KUKA KRL program: EPS_2_25862_MH02_A_20251016040656.src

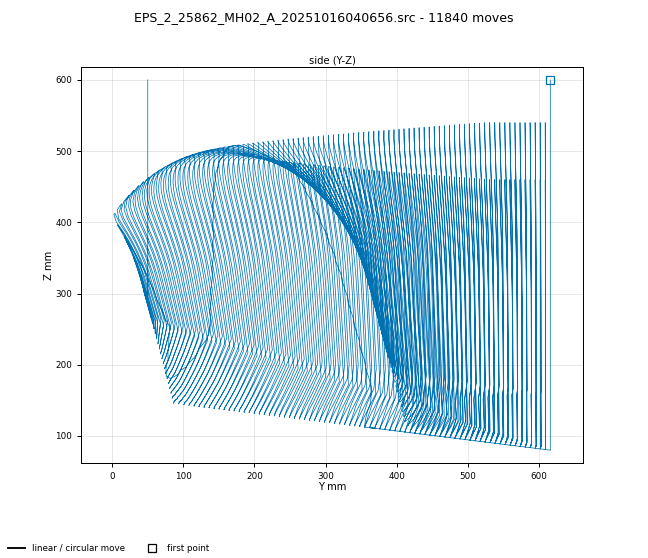
[picture p0: tool path of EPS_2_25862_MH02_A_20251016040656.src, 11840 of 11842 moves have a stored position in this frame; points joined in program order, loops and branches not executed]
&ACCESS RVP
&REL 4
&COMMENT QRS 19112012
&PARAM EDITMASK = *
DEF PART()
EXT BAS (BAS_COMMAND :IN,REAL :IN )
INT I
BAS (#INITMOV,0 )

;KUKA QRS Post kuka4.cps  Date:22-06-2017 !

File_ID=2894

QRS_PRE_INIT()

;Init var - Until changes are made in qrs_pre_init
Outlet_Square_prg=0
Inlet_1_Square_prg=0
Inlet_2_Square_prg=0
Inlet_3_Square_prg=0
Inlet_4_Square_prg=0
Inlet_5_Square_prg=0

Outlet_1={X 0.000, Y 524.050, Z 357.000, B 0.000, E1 0.000 }
Inlet_1={X 0.000, Y 530.010, Z 277.000, B 0.000, E1 270.000 }
Outlet_1_type=366
Inlet_1_type=366
;QRS#1=Sidecore dimensions
;QRS#2=375-15" PVC SDR 35
;QRS#3=375-15" PVC SDR 35
;QRS#4=
;QRS#5=
;QRS#6=
;QRS#7=
;QRS#8=
;QRS#9=20Y PSX
;QRS#10=20Y PSX
;QRS#11=
;QRS#12=
;QRS#13=
;QRS#14=
;QRS#15=
;QRS#16=1220x127x838 2,75'
;QRS#17=EPS Height
;QRS#18=540
;QRS#19=*
;QRS#20= UPDATED VERSION 22-06-2017
;QRS#21=*
Outlet_Square=0250
Inlet_1_Square=0250
Inlet_2_Square=0
Inlet_3_Square=0
Inlet_4_Square=0
Inlet_5_Square=0
Mill_Square=1
Outlet_Square_Prg=252
Inlet_1_Square_prg=252

QRS_INIT()

$ADVANCE=5

; T1
PTP {E1 173.606,E2 173.606}
PTP {X 0,Y 615.5,A -85,B 0,C 180,E1 173.606,E2 173.606,E3 0,E4 0,E5 0,E6 0}
QRS_SPEED_INIT()
LIN {X 0,Y 615.5,Z 600,A -85,B 0,C 180,E1 173.606,E2 173.606,E3 0,E4 0,E5 0,E6 0} C_VEL
LIN {X 0,Y 615.5,Z 90.176,A -85,B 0,C 180,E1 173.606,E2 173.606} C_VEL
LIN {X 0,Y 615.5,Z 81.996,A -85,B 0,C 180,E1 173.606,E2 173.606} C_VEL
LIN {X 0,Y 615.484,Z 79.996,A -85,B 0,C 180,E1 173.42,E2 173.42} C_VEL
LIN {X 0,Y 615.476,Z 80.009,A -85,B 0,C 180,E1 170.801,E2 170.801} C_VEL
LIN {X 0,Y 615.482,Z 80.003,A -85,B 0,C 180,E1 168.139,E2 168.139} C_VEL
LIN {X 0,Y 615.478,Z 79.998,A -85,B 0,C 180,E1 165.451,E2 165.451} C_VEL
LIN {X 0,Y 615.495,Z 80.012,A -85,B 0,C 180,E1 162.73,E2 162.73} C_VEL
LIN {X 0,Y 615.491,Z 79.995,A -85,B 0,C 180,E1 159.967,E2 159.967} C_VEL
LIN {X 0,Y 615.473,Z 80.006,A -85,B 0,C 180,E1 157.155,E2 157.155} C_VEL
LIN {X 0,Y 615.483,Z 80.004,A -85,B 0,C 180,E1 154.431,E2 154.431} C_VEL
LIN {X 0,Y 615.484,Z 79.997,A -85,B 0,C 180,E1 152.085,E2 152.085} C_VEL
LIN {X 0,Y 615.486,Z 79.995,A -85,B 0,C 180,E1 149.84,E2 149.84} C_VEL
LIN {X 0,Y 615.473,Z 80.002,A -85,B 0,C 180,E1 147.542,E2 147.542} C_VEL
LIN {X 0,Y 615.483,Z 80.009,A -85,B 0,C 180,E1 145.185,E2 145.185} C_VEL
LIN {X 0,Y 615.485,Z 80.007,A -85,B 0,C 180,E1 142.758,E2 142.758} C_VEL
LIN {X 0,Y 615.481,Z 79.997,A -85,B 0,C 180,E1 139.911,E2 139.911} C_VEL
LIN {X 0,Y 615.473,Z 80.003,A -85,B 0,C 180,E1 137.646,E2 137.646} C_VEL
LIN {X 0,Y 615.486,Z 80.008,A -85,B 0,C 180,E1 134.931,E2 134.931} C_VEL
LIN {X 0,Y 615.483,Z 79.996,A -85,B 0,C 180,E1 132.08,E2 132.08} C_VEL
LIN {X 0,Y 615.473,Z 80.003,A -85,B 0,C 180,E1 129.751,E2 129.751} C_VEL
LIN {X 0,Y 615.482,Z 80.005,A -85,B 0,C 180,E1 126.936,E2 126.936} C_VEL
LIN {X 0,Y 615.473,Z 80,A -85,B 0,C 180,E1 124.022,E2 124.022} C_VEL
LIN {X 0,Y 615.479,Z 80.007,A -85,B 0,C 180,E1 121.685,E2 121.685} C_VEL
LIN {X 0,Y 615.491,Z 80.014,A -85,B 0,C 180,E1 119.406,E2 119.406} C_VEL
LIN {X 0,Y 615.485,Z 79.995,A -85,B 0,C 180,E1 116.444,E2 116.444} C_VEL
LIN {X 0,Y 615.485,Z 80.015,A -85,B 0,C 180,E1 113.556,E2 113.556} C_VEL
LIN {X 0,Y 615.485,Z 79.996,A -85,B 0,C 180,E1 110.556,E2 110.556} C_VEL
LIN {X 0,Y 615.475,Z 80.007,A -85,B 0,C 180,E1 107.957,E2 107.957} C_VEL
LIN {X 0,Y 615.481,Z 80.003,A -85,B 0,C 180,E1 105.226,E2 105.226} C_VEL
LIN {X 0,Y 615.481,Z 79.997,A -85,B 0,C 180,E1 102.53,E2 102.53} C_VEL
LIN {X 0,Y 615.492,Z 80.011,A -85,B 0,C 180,E1 99.862,E2 99.862} C_VEL
LIN {X 0,Y 615.482,Z 80,A -85,B 0,C 180,E1 97.215,E2 97.215} C_VEL
LIN {X 0,Y 615.478,Z 79.999,A -85,B 0,C 180,E1 94.584,E2 94.584} C_VEL
LIN {X 0,Y 615.495,Z 80.012,A -85,B 0,C 180,E1 91.963,E2 91.963} C_VEL
LIN {X 0,Y 615.482,Z 79.999,A -85,B 0,C 180,E1 89.345,E2 89.345} C_VEL
LIN {X 0,Y 615.479,Z 79.999,A -85,B 0,C 180,E1 86.727,E2 86.727} C_VEL
LIN {X 0,Y 615.493,Z 80.012,A -85,B 0,C 180,E1 84.101,E2 84.101} C_VEL
LIN {X 0,Y 615.482,Z 79.999,A -85,B 0,C 180,E1 81.463,E2 81.463} C_VEL
LIN {X 0,Y 615.477,Z 80,A -85,B 0,C 180,E1 78.806,E2 78.806} C_VEL
LIN {X 0,Y 615.491,Z 80.01,A -85,B 0,C 180,E1 76.066,E2 76.066} C_VEL
LIN {X 0,Y 615.49,Z 79.995,A -85,B 0,C 180,E1 73.413,E2 73.413} C_VEL
LIN {X 0,Y 615.477,Z 80.005,A -85,B 0,C 180,E1 70.661,E2 70.661} C_VEL
LIN {X 0,Y 615.479,Z 80.003,A -85,B 0,C 180,E1 67.863,E2 67.863} C_VEL
LIN {X 0,Y 615.477,Z 80,A -85,B 0,C 180,E1 65.007,E2 65.007} C_VEL
LIN {X 0,Y 615.477,Z 80.005,A -85,B 0,C 180,E1 62.822,E2 62.822} C_VEL
LIN {X 0,Y 615.483,Z 80.007,A -85,B 0,C 180,E1 60.206,E2 60.206} C_VEL
LIN {X 0,Y 615.493,Z 79.994,A -85,B 0,C 180,E1 57.542,E2 57.542} C_VEL
LIN {X 0,Y 615.477,Z 80,A -85,B 0,C 180,E1 55.184,E2 55.184} C_VEL
LIN {X 0,Y 615.486,Z 80.01,A -85,B 0,C 180,E1 52.757,E2 52.757} C_VEL
LIN {X 0,Y 615.482,Z 79.998,A -85,B 0,C 180,E1 49.912,E2 49.912} C_VEL
LIN {X 0,Y 615.495,Z 79.993,A -85,B 0,C 180,E1 47.647,E2 47.647} C_VEL
LIN {X 0,Y 615.48,Z 80.01,A -85,B 0,C 180,E1 44.93,E2 44.93} C_VEL
LIN {X 0,Y 615.481,Z 79.998,A -85,B 0,C 180,E1 42.079,E2 42.079} C_VEL
LIN {X 0,Y 615.49,Z 79.995,A -85,B 0,C 180,E1 39.75,E2 39.75} C_VEL
LIN {X 0,Y 615.484,Z 80.014,A -85,B 0,C 180,E1 36.936,E2 36.936} C_VEL
LIN {X 0,Y 615.487,Z 79.995,A -85,B 0,C 180,E1 34.022,E2 34.022} C_VEL
LIN {X 0,Y 615.482,Z 80.012,A -85,B 0,C 180,E1 31.084,E2 31.084} C_VEL
LIN {X 0,Y 615.478,Z 80.001,A -85,B 0,C 180,E1 28.448,E2 28.448} C_VEL
LIN {X 0,Y 615.478,Z 80,A -85,B 0,C 180,E1 25.716,E2 25.716} C_VEL
LIN {X 0,Y 615.474,Z 80.004,A -85,B 0,C 180,E1 23.557,E2 23.557} C_VEL
LIN {X 0,Y 615.491,Z 80.049,A -85,B 0,C 180,E1 22.026,E2 22.026} C_VEL
LIN {X 0,Y 615.487,Z 80.696,A -85,B 0,C 180,E1 21.96,E2 21.96} C_VEL
LIN {X 0,Y 615.489,Z 286.31,A -85,B 0,C 180,E1 19.425,E2 19.425} C_VEL
LIN {X 0,Y 615.49,Z 302.93,A -85,B 0,C 180,E1 19.078,E2 19.078} C_VEL
LIN {X 0,Y 615.495,Z 319.071,A -85,B 0,C 180,E1 18.606,E2 18.606} C_VEL
LIN {X 0,Y 615.496,Z 334.183,A -85,B 0,C 180,E1 18.038,E2 18.038} C_VEL
LIN {X 0,Y 615.496,Z 348.835,A -85,B 0,C 180,E1 17.356,E2 17.356} C_VEL
LIN {X 0,Y 615.497,Z 363.769,A -85,B 0,C 180,E1 16.51,E2 16.51} C_VEL
LIN {X 0,Y 615.496,Z 377.743,A -85,B 0,C 180,E1 15.565,E2 15.565} C_VEL
LIN {X 0,Y 615.497,Z 390.512,A -85,B 0,C 180,E1 14.549,E2 14.549} C_VEL
LIN {X 0,Y 615.499,Z 401.486,A -85,B 0,C 180,E1 13.537,E2 13.537} C_VEL
LIN {X 0,Y 615.497,Z 412.376,A -85,B 0,C 180,E1 12.362,E2 12.362} C_VEL
LIN {X 0,Y 615.492,Z 422.792,A -85,B 0,C 180,E1 11.041,E2 11.041} C_VEL
LIN {X 0,Y 615.492,Z 431.704,A -85,B 0,C 180,E1 9.696,E2 9.696} C_VEL
LIN {X 0,Y 615.489,Z 438.268,A -85,B 0,C 180,E1 8.537,E2 8.537} C_VEL
LIN {X 0,Y 615.495,Z 445.804,A -85,B 0,C 180,E1 6.896,E2 6.896} C_VEL
LIN {X 0,Y 615.495,Z 451.596,A -85,B 0,C 180,E1 5.241,E2 5.241} C_VEL
LIN {X 0,Y 615.492,Z 454.979,A -85,B 0,C 180,E1 3.929,E2 3.929} C_VEL
LIN {X 0,Y 615.49,Z 457.428,A -85,B 0,C 180,E1 2.618,E2 2.618} C_VEL
LIN {X 0,Y 615.491,Z 458.838,A -85,B 0,C 180,E1 1.309,E2 1.309} C_VEL
LIN {X 0,Y 615.49,Z 459.385,A -85,B 0,C 180,E1 0,E2 0} C_VEL
LIN {X 0,Y 615.489,Z 458.902,A -85,B 0,C 180,E1 -1.309,E2 -1.309} C_VEL
LIN {X 0,Y 615.492,Z 457.568,A -85,B 0,C 180,E1 -2.618,E2 -2.618} C_VEL
LIN {X 0,Y 615.491,Z 455.174,A -85,B 0,C 180,E1 -3.928,E2 -3.928} C_VEL
LIN {X 0,Y 615.49,Z 451.879,A -85,B 0,C 180,E1 -5.241,E2 -5.241} C_VEL
LIN {X 0,Y 615.492,Z 446.153,A -85,B 0,C 180,E1 -6.898,E2 -6.898} C_VEL
LIN {X 0,Y 615.493,Z 440.328,A -85,B 0,C 180,E1 -8.206,E2 -8.206} C_VEL
LIN {X 0,Y 615.489,Z 432.251,A -85,B 0,C 180,E1 -9.696,E2 -9.696} C_VEL
LIN {X 0,Y 615.493,Z 423.461,A -85,B 0,C 180,E1 -11.041,E2 -11.041} C_VEL
LIN {X 0,Y 615.498,Z 413.171,A -85,B 0,C 180,E1 -12.362,E2 -12.362} C_VEL
LIN {X 0,Y 615.495,Z 402.356,A -85,B 0,C 180,E1 -13.537,E2 -13.537} C_VEL
LIN {X 0,Y 615.496,Z 391.545,A -85,B 0,C 180,E1 -14.549,E2 -14.549} C_VEL
LIN {X 0,Y 615.497,Z 377.814,A -85,B 0,C 180,E1 -15.65,E2 -15.65} C_VEL
LIN {X 0,Y 615.498,Z 363.993,A -85,B 0,C 180,E1 -16.586,E2 -16.586} C_VEL
LIN {X 0,Y 615.492,Z 348.926,A -85,B 0,C 180,E1 -17.442,E2 -17.442} C_VEL
LIN {X 0,Y 615.487,Z 332.529,A -85,B 0,C 180,E1 -18.2,E2 -18.2} C_VEL
LIN {X 0,Y 615.489,Z 316.698,A -85,B 0,C 180,E1 -18.775,E2 -18.775} C_VEL
LIN {X 0,Y 615.499,Z 301.255,A -85,B 0,C 180,E1 -19.207,E2 -19.207} C_VEL
LIN {X 0,Y 615.49,Z 285.06,A -85,B 0,C 180,E1 -19.533,E2 -19.533} C_VEL
LIN {X 0,Y 615.419,Z 80.715,A -85,B 0,C 180,E1 -22.051,E2 -22.051} C_VEL
LIN {X 0,Y 615.418,Z 80.012,A -85,B 0,C 180,E1 -22.139,E2 -22.139} C_VEL
LIN {X 0,Y 615.489,Z 80.013,A -85,B 0,C 180,E1 -24.992,E2 -24.992} C_VEL
LIN {X 0,Y 615.48,Z 80.009,A -85,B 0,C 180,E1 -27.177,E2 -27.177} C_VEL
LIN {X 0,Y 615.429,Z 80.01,A -85,B 0,C 180,E1 -29.784,E2 -29.784} C_VEL
LIN {X 0,Y 615.434,Z 80.008,A -85,B 0,C 180,E1 -31.688,E2 -31.688} C_VEL
LIN {X 0,Y 615.442,Z 80.009,A -85,B 0,C 180,E1 -34.025,E2 -34.025} C_VEL
LIN {X 0,Y 615.478,Z 80.014,A -85,B 0,C 180,E1 -36.425,E2 -36.425} C_VEL
LIN {X 0,Y 615.476,Z 80.001,A -85,B 0,C 180,E1 -39.06,E2 -39.06} C_VEL
LIN {X 0,Y 615.453,Z 80.005,A -85,B 0,C 180,E1 -41.476,E2 -41.476} C_VEL
LIN {X 0,Y 615.494,Z 80.014,A -85,B 0,C 180,E1 -44.149,E2 -44.149} C_VEL
LIN {X 0,Y 615.478,Z 79.998,A -85,B 0,C 180,E1 -46.953,E2 -46.953} C_VEL
LIN {X 0,Y 615.467,Z 80.005,A -85,B 0,C 180,E1 -49.392,E2 -49.392} C_VEL
LIN {X 0,Y 615.489,Z 80.008,A -85,B 0,C 180,E1 -51.988,E2 -51.988} C_VEL
LIN {X 0,Y 615.487,Z 79.998,A -85,B 0,C 180,E1 -54.384,E2 -54.384} C_VEL
LIN {X 0,Y 615.485,Z 79.997,A -85,B 0,C 180,E1 -56.763,E2 -56.763} C_VEL
LIN {X 0,Y 615.481,Z 80.005,A -85,B 0,C 180,E1 -59.08,E2 -59.08} C_VEL
LIN {X 0,Y 615.482,Z 80.01,A -85,B 0,C 180,E1 -61.55,E2 -61.55} C_VEL
LIN {X 0,Y 615.477,Z 80.197,A -85,B 0,C 180,E1 -62.153,E2 -62.153} C_VEL
LIN {X 0,Y 615.495,Z 116.189,A -85,B 0,C 180,E1 -64.864,E2 -64.864} C_VEL
LIN {X 0,Y 615.439,Z 150.773,A -85,B 0,C 180,E1 -67.409,E2 -67.409} C_VEL
LIN {X 0,Y 615.455,Z 158.788,A -85,B 0,C 180,E1 -67.972,E2 -67.972} C_VEL
LIN {X 0,Y 615.495,Z 366.404,A -85,B 0,C 180,E1 -70.532,E2 -70.532} C_VEL
LIN {X 0,Y 615.493,Z 382.979,A -85,B 0,C 180,E1 -70.878,E2 -70.878} C_VEL
LIN {X 0,Y 615.493,Z 397.921,A -85,B 0,C 180,E1 -71.311,E2 -71.311} C_VEL
LIN {X 0,Y 615.491,Z 413.342,A -85,B 0,C 180,E1 -71.88,E2 -71.88} C_VEL
LIN {X 0,Y 615.493,Z 427.997,A -85,B 0,C 180,E1 -72.558,E2 -72.558} C_VEL
LIN {X 0,Y 615.5,Z 441.829,A -85,B 0,C 180,E1 -73.328,E2 -73.328} C_VEL
LIN {X 0,Y 615.499,Z 456.032,A -85,B 0,C 180,E1 -74.265,E2 -74.265} C_VEL
LIN {X 0,Y 615.498,Z 469.087,A -85,B 0,C 180,E1 -75.282,E2 -75.282} C_VEL
LIN {X 0,Y 615.492,Z 480.209,A -85,B 0,C 180,E1 -76.294,E2 -76.294} C_VEL
LIN {X 0,Y 615.494,Z 491.287,A -85,B 0,C 180,E1 -77.47,E2 -77.47} C_VEL
LIN {X 0,Y 615.494,Z 500.763,A -85,B 0,C 180,E1 -78.64,E2 -78.64} C_VEL
LIN {X 0,Y 615.494,Z 509.962,A -85,B 0,C 180,E1 -79.971,E2 -79.971} C_VEL
LIN {X 0,Y 615.49,Z 518.499,A -85,B 0,C 180,E1 -81.463,E2 -81.463} C_VEL
LIN {X 0,Y 615.492,Z 525.981,A -85,B 0,C 180,E1 -83.102,E2 -83.102} C_VEL
LIN {X 0,Y 615.496,Z 531.739,A -85,B 0,C 180,E1 -84.758,E2 -84.758} C_VEL
LIN {X 0,Y 615.49,Z 535.076,A -85,B 0,C 180,E1 -86.071,E2 -86.071} C_VEL
LIN {X 0,Y 615.488,Z 537.503,A -85,B 0,C 180,E1 -87.382,E2 -87.382} C_VEL
LIN {X 0,Y 615.493,Z 538.869,A -85,B 0,C 180,E1 -88.691,E2 -88.691} C_VEL
LIN {X 0,Y 615.489,Z 539.39,A -85,B 0,C 180,E1 -90,E2 -90} C_VEL
LIN {X 0,Y 615.493,Z 538.869,A -85,B 0,C 180,E1 -91.308,E2 -91.308} C_VEL
LIN {X 0,Y 615.488,Z 537.504,A -85,B 0,C 180,E1 -92.617,E2 -92.617} C_VEL
LIN {X 0,Y 615.49,Z 535.078,A -85,B 0,C 180,E1 -93.928,E2 -93.928} C_VEL
LIN {X 0,Y 615.496,Z 531.742,A -85,B 0,C 180,E1 -95.241,E2 -95.241} C_VEL
LIN {X 0,Y 615.491,Z 525.983,A -85,B 0,C 180,E1 -96.898,E2 -96.898} C_VEL
LIN {X 0,Y 615.49,Z 518.504,A -85,B 0,C 180,E1 -98.536,E2 -98.536} C_VEL
LIN {X 0,Y 615.494,Z 509.967,A -85,B 0,C 180,E1 -100.028,E2 -100.028} C_VEL
LIN {X 0,Y 615.494,Z 500.77,A -85,B 0,C 180,E1 -101.359,E2 -101.359} C_VEL
LIN {X 0,Y 615.495,Z 491.295,A -85,B 0,C 180,E1 -102.529,E2 -102.529} C_VEL
LIN {X 0,Y 615.493,Z 480.219,A -85,B 0,C 180,E1 -103.705,E2 -103.705} C_VEL
LIN {X 0,Y 615.499,Z 468.12,A -85,B 0,C 180,E1 -104.802,E2 -104.802} C_VEL
LIN {X 0,Y 615.497,Z 454.884,A -85,B 0,C 180,E1 -105.819,E2 -105.819} C_VEL
LIN {X 0,Y 615.5,Z 441.844,A -85,B 0,C 180,E1 -106.671,E2 -106.671} C_VEL
LIN {X 0,Y 615.493,Z 428.015,A -85,B 0,C 180,E1 -107.441,E2 -107.441} C_VEL
LIN {X 0,Y 615.491,Z 413.357,A -85,B 0,C 180,E1 -108.119,E2 -108.119} C_VEL
LIN {X 0,Y 615.493,Z 397.948,A -85,B 0,C 180,E1 -108.688,E2 -108.688} C_VEL
LIN {X 0,Y 615.498,Z 381.192,A -85,B 0,C 180,E1 -109.164,E2 -109.164} C_VEL
LIN {X 0,Y 615.495,Z 364.975,A -85,B 0,C 180,E1 -109.489,E2 -109.489} C_VEL
LIN {X 0,Y 615.453,Z 158.208,A -85,B 0,C 180,E1 -112.049,E2 -112.049} C_VEL
LIN {X 0,Y 615.46,Z 124.216,A -85,B 0,C 180,E1 -114.542,E2 -114.542} C_VEL
LIN {X 0,Y 615.484,Z 89.011,A -85,B 0,C 180,E1 -117.177,E2 -117.177} C_VEL
LIN {X 0,Y 615.475,Z 79.998,A -85,B 0,C 180,E1 -117.869,E2 -117.869} C_VEL
LIN {X 0,Y 615.469,Z 80.004,A -85,B 0,C 180,E1 -120.161,E2 -120.161} C_VEL
LIN {X 0,Y 615.484,Z 80.01,A -85,B 0,C 180,E1 -122.457,E2 -122.457} C_VEL
LIN {X 0,Y 615.487,Z 80.008,A -85,B 0,C 180,E1 -124.814,E2 -124.814} C_VEL
LIN {X 0,Y 615.487,Z 79.997,A -85,B 0,C 180,E1 -127.242,E2 -127.242} C_VEL
LIN {X 0,Y 615.469,Z 80.006,A -85,B 0,C 180,E1 -130.087,E2 -130.087} C_VEL
LIN {X 0,Y 615.489,Z 80.011,A -85,B 0,C 180,E1 -132.352,E2 -132.352} C_VEL
LIN {X 0,Y 615.483,Z 79.998,A -85,B 0,C 180,E1 -135.068,E2 -135.068} C_VEL
LIN {X 0,Y 615.471,Z 80.005,A -85,B 0,C 180,E1 -137.921,E2 -137.921} C_VEL
LIN {X 0,Y 615.493,Z 80.011,A -85,B 0,C 180,E1 -140.251,E2 -140.251} C_VEL
LIN {X 0,Y 615.485,Z 79.996,A -85,B 0,C 180,E1 -143.063,E2 -143.063} C_VEL
LIN {X 0,Y 615.482,Z 79.996,A -85,B 0,C 180,E1 -145.299,E2 -145.299} C_VEL
LIN {X 0,Y 615.467,Z 80.004,A -85,B 0,C 180,E1 -147.671,E2 -147.671} C_VEL
LIN {X 0,Y 615.496,Z 80.011,A -85,B 0,C 180,E1 -150.203,E2 -150.203} C_VEL
LIN {X 0,Y 615.497,Z 79.993,A -85,B 0,C 180,E1 -152.952,E2 -152.952} C_VEL
LIN {X 0,Y 615.476,Z 80.007,A -85,B 0,C 180,E1 -155.728,E2 -155.728} C_VEL
LIN {X 0,Y 615.483,Z 80,A -85,B 0,C 180,E1 -158.568,E2 -158.568} C_VEL
LIN {X 0,Y 615.47,Z 80.003,A -85,B 0,C 180,E1 -161.398,E2 -161.398} C_VEL
LIN {X 0,Y 615.489,Z 80.008,A -85,B 0,C 180,E1 -164.095,E2 -164.095} C_VEL
LIN {X 0,Y 615.493,Z 79.994,A -85,B 0,C 180,E1 -166.799,E2 -166.799} C_VEL
LIN {X 0,Y 615.473,Z 80.007,A -85,B 0,C 180,E1 -169.473,E2 -169.473} C_VEL
LIN {X 0,Y 615.484,Z 80.004,A -85,B 0,C 180,E1 -172.124,E2 -172.124} C_VEL
LIN {X 0,Y 615.485,Z 79.995,A -85,B 0,C 180,E1 -174.759,E2 -174.759} C_VEL
LIN {X 0,Y 615.478,Z 80.007,A -85,B 0,C 180,E1 -177.382,E2 -177.382} C_VEL
LIN {X 0,Y 615.483,Z 80.004,A -85,B 0,C 180,E1 -180,E2 -180} C_VEL
LIN {X 0,Y 615.486,Z 79.995,A -85,B 0,C 180,E1 -182.618,E2 -182.618} C_VEL
LIN {X 0,Y 615.474,Z 80.008,A -85,B 0,C 180,E1 -185.241,E2 -185.241} C_VEL
LIN {X 0,Y 615.484,Z 79.996,A -85,B 0,C 180,E1 -186.58,E2 -186.58} C_VEL
LIN {X 0,Y 614.804,Z 80.154,A -85,B 0,C 180,E1 -187.126,E2 -187.126} C_VEL
LIN {X 0,Y 611.965,Z 80.565,A -85,B 0,C 180,E1 -188.012,E2 -188.012} C_VEL
LIN {X 0,Y 609.573,Z 80.879,A -85,B 0,C 180,E1 -188.725,E2 -188.725} C_VEL
LIN {X 0,Y 608.54,Z 80.998,A -85,B 0,C 180,E1 -189.275,E2 -189.275} C_VEL
LIN {X 0,Y 608.452,Z 81.006,A -85,B 0,C 180,E1 -189.461,E2 -189.461} C_VEL
LIN {X 0,Y 608.458,Z 81.001,A -85,B 0,C 180,E1 -192,E2 -192} C_VEL
LIN {X 0,Y 608.469,Z 80.999,A -85,B 0,C 180,E1 -194.721,E2 -194.721} C_VEL
LIN {X 0,Y 608.456,Z 81.007,A -85,B 0,C 180,E1 -197.476,E2 -197.476} C_VEL
LIN {X 0,Y 608.459,Z 80.999,A -85,B 0,C 180,E1 -200.274,E2 -200.274} C_VEL
LIN {X 0,Y 608.454,Z 81,A -85,B 0,C 180,E1 -202.477,E2 -202.477} C_VEL
LIN {X 0,Y 608.451,Z 81.001,A -85,B 0,C 180,E1 -204.571,E2 -204.571} C_VEL
LIN {X 0,Y 608.48,Z 81.006,A -85,B 0,C 180,E1 -207.209,E2 -207.209} C_VEL
LIN {X 0,Y 608.468,Z 80.998,A -85,B 0,C 180,E1 -209.973,E2 -209.973} C_VEL
LIN {X 0,Y 608.45,Z 81.003,A -85,B 0,C 180,E1 -212.522,E2 -212.522} C_VEL
LIN {X 0,Y 608.441,Z 81.007,A -85,B 0,C 180,E1 -215.278,E2 -215.278} C_VEL
LIN {X 0,Y 608.467,Z 80.999,A -85,B 0,C 180,E1 -217.746,E2 -217.746} C_VEL
LIN {X 0,Y 608.445,Z 81.003,A -85,B 0,C 180,E1 -220.329,E2 -220.329} C_VEL
LIN {X 0,Y 608.47,Z 81.001,A -85,B 0,C 180,E1 -223.31,E2 -223.31} C_VEL
LIN {X 0,Y 608.467,Z 80.999,A -85,B 0,C 180,E1 -226.131,E2 -226.131} C_VEL
LIN {X 0,Y 608.454,Z 81.01,A -85,B 0,C 180,E1 -228.824,E2 -228.824} C_VEL
LIN {X 0,Y 608.465,Z 80.999,A -85,B 0,C 180,E1 -231.412,E2 -231.412} C_VEL
LIN {X 0,Y 608.442,Z 81.002,A -85,B 0,C 180,E1 -233.955,E2 -233.955} C_VEL
LIN {X 0,Y 608.463,Z 81.004,A -85,B 0,C 180,E1 -236.33,E2 -236.33} C_VEL
LIN {X 0,Y 608.458,Z 81.008,A -85,B 0,C 180,E1 -238.731,E2 -238.731} C_VEL
LIN {X 0,Y 608.473,Z 80.998,A -85,B 0,C 180,E1 -241.38,E2 -241.38} C_VEL
LIN {X 0,Y 608.472,Z 81.004,A -85,B 0,C 180,E1 -244.279,E2 -244.279} C_VEL
LIN {X 0,Y 608.449,Z 81.004,A -85,B 0,C 180,E1 -246.877,E2 -246.877} C_VEL
LIN {X 0,Y 608.466,Z 80.998,A -85,B 0,C 180,E1 -249.322,E2 -249.322} C_VEL
LIN {X 0,Y 608.442,Z 81.003,A -85,B 0,C 180,E1 -251.828,E2 -251.828} C_VEL
LIN {X 0,Y 608.466,Z 81.004,A -85,B 0,C 180,E1 -254.594,E2 -254.594} C_VEL
LIN {X 0,Y 608.471,Z 80.998,A -85,B 0,C 180,E1 -257.323,E2 -257.323} C_VEL
LIN {X 0,Y 608.46,Z 81.006,A -85,B 0,C 180,E1 -260.023,E2 -260.023} C_VEL
LIN {X 0,Y 608.462,Z 81.001,A -85,B 0,C 180,E1 -262.701,E2 -262.701} C_VEL
LIN {X 0,Y 608.447,Z 81.001,A -85,B 0,C 180,E1 -265.363,E2 -265.363} C_VEL
LIN {X 0,Y 608.464,Z 81.008,A -85,B 0,C 180,E1 -268.015,E2 -268.015} C_VEL
LIN {X 0,Y 608.477,Z 80.999,A -85,B 0,C 180,E1 -270.662,E2 -270.662} C_VEL
LIN {X 0,Y 608.473,Z 80.998,A -85,B 0,C 180,E1 -273.311,E2 -273.311} C_VEL
LIN {X 0,Y 608.466,Z 81.009,A -85,B 0,C 180,E1 -275.967,E2 -275.967} C_VEL
LIN {X 0,Y 608.452,Z 81.001,A -85,B 0,C 180,E1 -278.636,E2 -278.636} C_VEL
LIN {X 0,Y 608.456,Z 81.002,A -85,B 0,C 180,E1 -281.325,E2 -281.325} C_VEL
LIN {X 0,Y 608.471,Z 81.004,A -85,B 0,C 180,E1 -284.038,E2 -284.038} C_VEL
LIN {X 0,Y 608.476,Z 80.997,A -85,B 0,C 180,E1 -286.784,E2 -286.784} C_VEL
LIN {X 0,Y 608.446,Z 81.009,A -85,B 0,C 180,E1 -289.571,E2 -289.571} C_VEL
LIN {X 0,Y 608.479,Z 80.997,A -85,B 0,C 180,E1 -292.406,E2 -292.406} C_VEL
LIN {X 0,Y 608.45,Z 81.005,A -85,B 0,C 180,E1 -295.301,E2 -295.301} C_VEL
LIN {X 0,Y 608.445,Z 81.011,A -85,B 0,C 180,E1 -297.519,E2 -297.519} C_VEL
LIN {X 0,Y 608.464,Z 81.002,A -85,B 0,C 180,E1 -299.971,E2 -299.971} C_VEL
LIN {X 0,Y 608.457,Z 81.001,A -85,B 0,C 180,E1 -302.88,E2 -302.88} C_VEL
LIN {X 0,Y 608.441,Z 81.009,A -85,B 0,C 180,E1 -305.278,E2 -305.278} C_VEL
LIN {X 0,Y 608.466,Z 81.003,A -85,B 0,C 180,E1 -307.747,E2 -307.747} C_VEL
LIN {X 0,Y 608.447,Z 81.001,A -85,B 0,C 180,E1 -310.329,E2 -310.329} C_VEL
LIN {X 0,Y 608.481,Z 81.007,A -85,B 0,C 180,E1 -313.31,E2 -313.31} C_VEL
LIN {X 0,Y 608.469,Z 80.998,A -85,B 0,C 180,E1 -316.131,E2 -316.131} C_VEL
LIN {X 0,Y 608.45,Z 81.004,A -85,B 0,C 180,E1 -318.823,E2 -318.823} C_VEL
LIN {X 0,Y 608.466,Z 81,A -85,B 0,C 180,E1 -321.76,E2 -321.76} C_VEL
LIN {X 0,Y 608.464,Z 80.999,A -85,B 0,C 180,E1 -323.953,E2 -323.953} C_VEL
LIN {X 0,Y 608.448,Z 81.001,A -85,B 0,C 180,E1 -326.328,E2 -326.328} C_VEL
LIN {X 0,Y 608.448,Z 81.006,A -85,B 0,C 180,E1 -328.733,E2 -328.733} C_VEL
LIN {X 0,Y 608.468,Z 81.002,A -85,B 0,C 180,E1 -331.382,E2 -331.382} C_VEL
LIN {X 0,Y 608.437,Z 81.002,A -85,B 0,C 180,E1 -333.964,E2 -333.964} C_VEL
LIN {X 0,Y 608.467,Z 80.999,A -85,B 0,C 180,E1 -336.155,E2 -336.155} C_VEL
LIN {X 0,Y 608.469,Z 80.999,A -85,B 0,C 180,E1 -337.773,E2 -337.773} C_VEL
LIN {X 0,Y 608.912,Z 84.157,A -85,B 0,C 180,E1 -337.835,E2 -337.835} C_VEL
LIN {X 0,Y 608.817,Z 284.856,A -85,B 0,C 180,E1 -340.332,E2 -340.332} C_VEL
LIN {X 0,Y 608.794,Z 301.155,A -85,B 0,C 180,E1 -340.66,E2 -340.66} C_VEL
LIN {X 0,Y 608.756,Z 316.608,A -85,B 0,C 180,E1 -341.096,E2 -341.096} C_VEL
LIN {X 0,Y 608.704,Z 332.317,A -85,B 0,C 180,E1 -341.672,E2 -341.672} C_VEL
LIN {X 0,Y 608.67,Z 347.11,A -85,B 0,C 180,E1 -342.356,E2 -342.356} C_VEL
LIN {X 0,Y 608.618,Z 361.108,A -85,B 0,C 180,E1 -343.134,E2 -343.134} C_VEL
LIN {X 0,Y 608.579,Z 375.441,A -85,B 0,C 180,E1 -344.081,E2 -344.081} C_VEL
LIN {X 0,Y 608.558,Z 388.606,A -85,B 0,C 180,E1 -345.11,E2 -345.11} C_VEL
LIN {X 0,Y 608.515,Z 401.57,A -85,B 0,C 180,E1 -346.304,E2 -346.304} C_VEL
LIN {X 0,Y 608.493,Z 412.517,A -85,B 0,C 180,E1 -347.493,E2 -347.493} C_VEL
LIN {X 0,Y 608.491,Z 421.878,A -85,B 0,C 180,E1 -348.676,E2 -348.676} C_VEL
LIN {X 0,Y 608.466,Z 430.986,A -85,B 0,C 180,E1 -350.023,E2 -350.023} C_VEL
LIN {X 0,Y 608.445,Z 438.616,A -85,B 0,C 180,E1 -351.364,E2 -351.364} C_VEL
LIN {X 0,Y 608.456,Z 444.858,A -85,B 0,C 180,E1 -352.7,E2 -352.7} C_VEL
LIN {X 0,Y 608.431,Z 449.98,A -85,B 0,C 180,E1 -354.033,E2 -354.033} C_VEL
LIN {X 0,Y 608.429,Z 453.936,A -85,B 0,C 180,E1 -355.362,E2 -355.362} C_VEL
LIN {X 0,Y 608.423,Z 456.906,A -85,B 0,C 180,E1 -356.689,E2 -356.689} C_VEL
LIN {X 0,Y 608.432,Z 458.836,A -85,B 0,C 180,E1 -358.014,E2 -358.014} C_VEL
LIN {X 0,Y 608.438,Z 459.84,A -85,B 0,C 180,E1 -359.338,E2 -359.338} C_VEL
LIN {X 0,Y 608.439,Z 459.861,A -85,B 0,C 180,E1 -360.662,E2 -360.662} C_VEL
LIN {X 0,Y 608.431,Z 458.942,A -85,B 0,C 180,E1 -361.986,E2 -361.986} C_VEL
LIN {X 0,Y 608.422,Z 457.056,A -85,B 0,C 180,E1 -363.311,E2 -363.311} C_VEL
LIN {X 0,Y 608.427,Z 454.177,A -85,B 0,C 180,E1 -364.638,E2 -364.638} C_VEL
LIN {X 0,Y 608.427,Z 450.267,A -85,B 0,C 180,E1 -365.967,E2 -365.967} C_VEL
LIN {X 0,Y 608.441,Z 445.243,A -85,B 0,C 180,E1 -367.3,E2 -367.3} C_VEL
LIN {X 0,Y 608.444,Z 439.086,A -85,B 0,C 180,E1 -368.636,E2 -368.636} C_VEL
LIN {X 0,Y 608.457,Z 430.516,A -85,B 0,C 180,E1 -370.145,E2 -370.145} C_VEL
LIN {X 0,Y 608.467,Z 421.301,A -85,B 0,C 180,E1 -371.493,E2 -371.493} C_VEL
LIN {X 0,Y 608.496,Z 410.329,A -85,B 0,C 180,E1 -372.846,E2 -372.846} C_VEL
LIN {X 0,Y 608.523,Z 398.977,A -85,B 0,C 180,E1 -374.036,E2 -374.036} C_VEL
LIN {X 0,Y 608.548,Z 386.592,A -85,B 0,C 180,E1 -375.147,E2 -375.147} C_VEL
LIN {X 0,Y 608.607,Z 374.336,A -85,B 0,C 180,E1 -376.09,E2 -376.09} C_VEL
LIN {X 0,Y 608.623,Z 359.755,A -85,B 0,C 180,E1 -377.038,E2 -377.038} C_VEL
LIN {X 0,Y 608.658,Z 345.432,A -85,B 0,C 180,E1 -377.817,E2 -377.817} C_VEL
LIN {X 0,Y 608.716,Z 330.428,A -85,B 0,C 180,E1 -378.492,E2 -378.492} C_VEL
LIN {X 0,Y 608.758,Z 314.04,A -85,B 0,C 180,E1 -379.078,E2 -379.078} C_VEL
LIN {X 0,Y 608.795,Z 296.666,A -85,B 0,C 180,E1 -379.537,E2 -379.537} C_VEL
LIN {X 0,Y 608.796,Z 280.502,A -85,B 0,C 180,E1 -379.822,E2 -379.822} C_VEL
LIN {X 0,Y 608.855,Z 84.226,A -85,B 0,C 180,E1 -382.256,E2 -382.256} C_VEL
LIN {X 0,Y 608.407,Z 81.008,A -85,B 0,C 180,E1 -382.318,E2 -382.318} C_VEL
LIN {X 0,Y 608.422,Z 81.007,A -85,B 0,C 180,E1 -384.572,E2 -384.572} C_VEL
LIN {X 0,Y 608.423,Z 81.006,A -85,B 0,C 180,E1 -387.519,E2 -387.519} C_VEL
LIN {X 0,Y 608.4,Z 81.007,A -85,B 0,C 180,E1 -389.96,E2 -389.96} C_VEL
LIN {X 0,Y 608.446,Z 81.008,A -85,B 0,C 180,E1 -392.52,E2 -392.52} C_VEL
LIN {X 0,Y 608.423,Z 81.005,A -85,B 0,C 180,E1 -395.279,E2 -395.279} C_VEL
LIN {X 0,Y 608.445,Z 81.002,A -85,B 0,C 180,E1 -397.748,E2 -397.748} C_VEL
LIN {X 0,Y 608.445,Z 81.012,A -85,B 0,C 180,E1 -400.328,E2 -400.328} C_VEL
LIN {X 0,Y 608.443,Z 81.002,A -85,B 0,C 180,E1 -402.96,E2 -402.96} C_VEL
LIN {X 0,Y 608.448,Z 81.006,A -85,B 0,C 180,E1 -405.737,E2 -405.737} C_VEL
LIN {X 0,Y 608.468,Z 81.008,A -85,B 0,C 180,E1 -407.939,E2 -407.939} C_VEL
LIN {X 0,Y 608.441,Z 81.002,A -85,B 0,C 180,E1 -410.706,E2 -410.706} C_VEL
LIN {X 0,Y 608.445,Z 81.003,A -85,B 0,C 180,E1 -413.084,E2 -413.084} C_VEL
LIN {X 0,Y 608.464,Z 81.008,A -85,B 0,C 180,E1 -415.53,E2 -415.53} C_VEL
LIN {X 0,Y 608.469,Z 81.003,A -85,B 0,C 180,E1 -417.905,E2 -417.905} C_VEL
LIN {X 0,Y 608.461,Z 81,A -85,B 0,C 180,E1 -420.22,E2 -420.22} C_VEL
LIN {X 0,Y 608.476,Z 81.107,A -85,B 0,C 180,E1 -421.875,E2 -421.875} C_VEL
LIN {X 0,Y 608.925,Z 84.142,A -85,B 0,C 180,E1 -422.132,E2 -422.132} C_VEL
LIN {X 0,Y 608.826,Z 121.776,A -85,B 0,C 180,E1 -424.989,E2 -424.989} C_VEL
LIN {X 0,Y 608.696,Z 155.171,A -85,B 0,C 180,E1 -427.469,E2 -427.469} C_VEL
LIN {X 0,Y 608.76,Z 158.788,A -85,B 0,C 180,E1 -427.717,E2 -427.717} C_VEL
LIN {X 0,Y 608.783,Z 294.163,A -85,B 0,C 180,E1 -429.399,E2 -429.399} C_VEL
LIN {X 0,Y 608.806,Z 366.403,A -85,B 0,C 180,E1 -430.309,E2 -430.309} C_VEL
LIN {X 0,Y 608.779,Z 382.98,A -85,B 0,C 180,E1 -430.659,E2 -430.659} C_VEL
LIN {X 0,Y 608.743,Z 399.217,A -85,B 0,C 180,E1 -431.139,E2 -431.139} C_VEL
LIN {X 0,Y 608.688,Z 415.204,A -85,B 0,C 180,E1 -431.753,E2 -431.753} C_VEL
LIN {X 0,Y 608.681,Z 429.722,A -85,B 0,C 180,E1 -432.443,E2 -432.443} C_VEL
LIN {X 0,Y 608.633,Z 444.927,A -85,B 0,C 180,E1 -433.324,E2 -433.324} C_VEL
LIN {X 0,Y 608.574,Z 458.363,A -85,B 0,C 180,E1 -434.253,E2 -434.253} C_VEL
LIN {X 0,Y 608.551,Z 471.063,A -85,B 0,C 180,E1 -435.281,E2 -435.281} C_VEL
LIN {X 0,Y 608.496,Z 483.63,A -85,B 0,C 180,E1 -436.474,E2 -436.474} C_VEL
LIN {X 0,Y 608.47,Z 494.327,A -85,B 0,C 180,E1 -437.661,E2 -437.661} C_VEL
LIN {X 0,Y 608.475,Z 504.861,A -85,B 0,C 180,E1 -439.04,E2 -439.04} C_VEL
LIN {X 0,Y 608.466,Z 513.281,A -85,B 0,C 180,E1 -440.358,E2 -440.358} C_VEL
LIN {X 0,Y 608.45,Z 520.484,A -85,B 0,C 180,E1 -441.698,E2 -441.698} C_VEL
LIN {X 0,Y 608.437,Z 526.467,A -85,B 0,C 180,E1 -443.033,E2 -443.033} C_VEL
LIN {X 0,Y 608.438,Z 532.244,A -85,B 0,C 180,E1 -444.697,E2 -444.697} C_VEL
LIN {X 0,Y 608.428,Z 535.632,A -85,B 0,C 180,E1 -446.025,E2 -446.025} C_VEL
LIN {X 0,Y 608.415,Z 538.085,A -85,B 0,C 180,E1 -447.351,E2 -447.351} C_VEL
LIN {X 0,Y 608.445,Z 539.477,A -85,B 0,C 180,E1 -448.676,E2 -448.676} C_VEL
LIN {X 0,Y 608.429,Z 540,A -85,B 0,C 180,E1 -450,E2 -450} C_VEL
LIN {X 0,Y 608.445,Z 539.477,A -85,B 0,C 180,E1 -451.323,E2 -451.323} C_VEL
LIN {X 0,Y 608.415,Z 538.086,A -85,B 0,C 180,E1 -452.648,E2 -452.648} C_VEL
LIN {X 0,Y 608.428,Z 535.633,A -85,B 0,C 180,E1 -453.974,E2 -453.974} C_VEL
LIN {X 0,Y 608.438,Z 532.247,A -85,B 0,C 180,E1 -455.302,E2 -455.302} C_VEL
LIN {X 0,Y 608.437,Z 526.47,A -85,B 0,C 180,E1 -456.966,E2 -456.966} C_VEL
LIN {X 0,Y 608.445,Z 518.86,A -85,B 0,C 180,E1 -458.636,E2 -458.636} C_VEL
LIN {X 0,Y 608.459,Z 510.248,A -85,B 0,C 180,E1 -460.145,E2 -460.145} C_VEL
LIN {X 0,Y 608.465,Z 500.971,A -85,B 0,C 180,E1 -461.492,E2 -461.492} C_VEL
LIN {X 0,Y 608.492,Z 491.426,A -85,B 0,C 180,E1 -462.676,E2 -462.676} C_VEL
LIN {X 0,Y 608.519,Z 479.972,A -85,B 0,C 180,E1 -463.896,E2 -463.896} C_VEL
LIN {X 0,Y 608.554,Z 468.148,A -85,B 0,C 180,E1 -464.975,E2 -464.975} C_VEL
LIN {X 0,Y 608.598,Z 454.892,A -85,B 0,C 180,E1 -466.004,E2 -466.004} C_VEL
LIN {X 0,Y 608.617,Z 441.848,A -85,B 0,C 180,E1 -466.865,E2 -466.865} C_VEL
LIN {X 0,Y 608.678,Z 426.271,A -85,B 0,C 180,E1 -467.73,E2 -467.73} C_VEL
LIN {X 0,Y 608.711,Z 411.377,A -85,B 0,C 180,E1 -468.41,E2 -468.41} C_VEL
LIN {X 0,Y 608.736,Z 395.362,A -85,B 0,C 180,E1 -468.991,E2 -468.991} C_VEL
LIN {X 0,Y 608.796,Z 379.369,A -85,B 0,C 180,E1 -469.427,E2 -469.427} C_VEL
LIN {X 0,Y 608.809,Z 363.469,A -85,B 0,C 180,E1 -469.734,E2 -469.734} C_VEL
LIN {X 0,Y 608.894,Z 159.759,A -85,B 0,C 180,E1 -472.266,E2 -472.266} C_VEL
LIN {X 0,Y 608.689,Z 158.208,A -85,B 0,C 180,E1 -472.307,E2 -472.307} C_VEL
LIN {X 0,Y 608.788,Z 125.43,A -85,B 0,C 180,E1 -474.738,E2 -474.738} C_VEL
LIN {X 0,Y 608.89,Z 91.787,A -85,B 0,C 180,E1 -477.283,E2 -477.283} C_VEL
LIN {X 0,Y 608.914,Z 82.941,A -85,B 0,C 180,E1 -477.962,E2 -477.962} C_VEL
LIN {X 0,Y 608.455,Z 81.005,A -85,B 0,C 180,E1 -478.149,E2 -478.149} C_VEL
LIN {X 0,Y 608.464,Z 81.008,A -85,B 0,C 180,E1 -480.545,E2 -480.545} C_VEL
LIN {X 0,Y 608.458,Z 81.006,A -85,B 0,C 180,E1 -482.879,E2 -482.879} C_VEL
LIN {X 0,Y 608.441,Z 81.002,A -85,B 0,C 180,E1 -485.277,E2 -485.277} C_VEL
LIN {X 0,Y 608.457,Z 81,A -85,B 0,C 180,E1 -487.746,E2 -487.746} C_VEL
LIN {X 0,Y 608.445,Z 81.009,A -85,B 0,C 180,E1 -490.329,E2 -490.329} C_VEL
LIN {X 0,Y 608.482,Z 80.996,A -85,B 0,C 180,E1 -493.31,E2 -493.31} C_VEL
LIN {X 0,Y 608.46,Z 81.005,A -85,B 0,C 180,E1 -496.13,E2 -496.13} C_VEL
LIN {X 0,Y 608.456,Z 81.002,A -85,B 0,C 180,E1 -498.824,E2 -498.824} C_VEL
LIN {X 0,Y 608.468,Z 80.998,A -85,B 0,C 180,E1 -501.412,E2 -501.412} C_VEL
LIN {X 0,Y 608.456,Z 81.005,A -85,B 0,C 180,E1 -503.952,E2 -503.952} C_VEL
LIN {X 0,Y 608.461,Z 81.008,A -85,B 0,C 180,E1 -506.329,E2 -506.329} C_VEL
LIN {X 0,Y 608.474,Z 80.999,A -85,B 0,C 180,E1 -508.727,E2 -508.727} C_VEL
LIN {X 0,Y 608.461,Z 80.999,A -85,B 0,C 180,E1 -511.381,E2 -511.381} C_VEL
LIN {X 0,Y 608.44,Z 81.01,A -85,B 0,C 180,E1 -513.964,E2 -513.964} C_VEL
LIN {X 0,Y 608.467,Z 81.007,A -85,B 0,C 180,E1 -516.155,E2 -516.155} C_VEL
LIN {X 0,Y 608.467,Z 81.004,A -85,B 0,C 180,E1 -518.309,E2 -518.309} C_VEL
LIN {X 0,Y 608.459,Z 81,A -85,B 0,C 180,E1 -521.286,E2 -521.286} C_VEL
LIN {X 0,Y 608.458,Z 81.01,A -85,B 0,C 180,E1 -523.906,E2 -523.906} C_VEL
LIN {X 0,Y 608.468,Z 80.998,A -85,B 0,C 180,E1 -526.644,E2 -526.644} C_VEL
LIN {X 0,Y 608.452,Z 81.003,A -85,B 0,C 180,E1 -529.35,E2 -529.35} C_VEL
LIN {X 0,Y 608.474,Z 81.003,A -85,B 0,C 180,E1 -532.033,E2 -532.033} C_VEL
LIN {X 0,Y 608.464,Z 80.998,A -85,B 0,C 180,E1 -534.698,E2 -534.698} C_VEL
LIN {X 0,Y 608.469,Z 81.003,A -85,B 0,C 180,E1 -537.352,E2 -537.352} C_VEL
LIN {X 0,Y 608.474,Z 81.002,A -85,B 0,C 180,E1 -540,E2 -540} C_VEL
LIN {X 0,Y 608.476,Z 80.997,A -85,B 0,C 180,E1 -542.648,E2 -542.648} C_VEL
LIN {X 0,Y 608.454,Z 81.006,A -85,B 0,C 180,E1 -545.302,E2 -545.302} C_VEL
LIN {X 0,Y 608.474,Z 81,A -85,B 0,C 180,E1 -547.967,E2 -547.967} C_VEL
LIN {X 0,Y 608.452,Z 81.006,A -85,B 0,C 180,E1 -549.461,E2 -549.461} C_VEL
LIN {X 0,Y 607.776,Z 81.087,A -85,B 0,C 180,E1 -550.013,E2 -550.013} C_VEL
LIN {X 0,Y 604.923,Z 81.442,A -85,B 0,C 180,E1 -550.91,E2 -550.91} C_VEL
LIN {X 0,Y 602.52,Z 81.746,A -85,B 0,C 180,E1 -551.632,E2 -551.632} C_VEL
LIN {X 0,Y 601.489,Z 81.868,A -85,B 0,C 180,E1 -552.189,E2 -552.189} C_VEL
LIN {X 0,Y 601.405,Z 81.878,A -85,B 0,C 180,E1 -552.377,E2 -552.377} C_VEL
LIN {X 0,Y 601.424,Z 81.878,A -85,B 0,C 180,E1 -554.897,E2 -554.897} C_VEL
LIN {X 0,Y 601.43,Z 81.879,A -85,B 0,C 180,E1 -556.986,E2 -556.986} C_VEL
LIN {X 0,Y 601.406,Z 81.88,A -85,B 0,C 180,E1 -559.809,E2 -559.809} C_VEL
LIN {X 0,Y 601.407,Z 81.88,A -85,B 0,C 180,E1 -562.683,E2 -562.683} C_VEL
LIN {X 0,Y 601.4,Z 81.884,A -85,B 0,C 180,E1 -564.879,E2 -564.879} C_VEL
LIN {X 0,Y 601.417,Z 81.877,A -85,B 0,C 180,E1 -567.868,E2 -567.868} C_VEL
LIN {X 0,Y 601.425,Z 81.875,A -85,B 0,C 180,E1 -570.164,E2 -570.164} C_VEL
LIN {X 0,Y 601.413,Z 81.881,A -85,B 0,C 180,E1 -572.715,E2 -572.715} C_VEL
LIN {X 0,Y 601.408,Z 81.886,A -85,B 0,C 180,E1 -575.115,E2 -575.115} C_VEL
LIN {X 0,Y 601.432,Z 81.878,A -85,B 0,C 180,E1 -577.419,E2 -577.419} C_VEL
LIN {X 0,Y 601.409,Z 81.877,A -85,B 0,C 180,E1 -579.995,E2 -579.995} C_VEL
LIN {X 0,Y 601.408,Z 81.884,A -85,B 0,C 180,E1 -582.671,E2 -582.671} C_VEL
LIN {X 0,Y 601.423,Z 81.877,A -85,B 0,C 180,E1 -585.482,E2 -585.482} C_VEL
LIN {X 0,Y 601.422,Z 81.88,A -85,B 0,C 180,E1 -588.407,E2 -588.407} C_VEL
LIN {X 0,Y 601.432,Z 81.883,A -85,B 0,C 180,E1 -590.876,E2 -590.876} C_VEL
LIN {X 0,Y 601.4,Z 81.879,A -85,B 0,C 180,E1 -593.418,E2 -593.418} C_VEL
LIN {X 0,Y 601.429,Z 81.877,A -85,B 0,C 180,E1 -596.065,E2 -596.065} C_VEL
LIN {X 0,Y 601.439,Z 81.883,A -85,B 0,C 180,E1 -598.542,E2 -598.542} C_VEL
LIN {X 0,Y 601.432,Z 81.875,A -85,B 0,C 180,E1 -601.374,E2 -601.374} C_VEL
LIN {X 0,Y 601.401,Z 81.878,A -85,B 0,C 180,E1 -603.637,E2 -603.637} C_VEL
LIN {X 0,Y 601.417,Z 81.885,A -85,B 0,C 180,E1 -606.59,E2 -606.59} C_VEL
LIN {X 0,Y 601.429,Z 81.875,A -85,B 0,C 180,E1 -609.479,E2 -609.479} C_VEL
LIN {X 0,Y 601.392,Z 81.889,A -85,B 0,C 180,E1 -612.312,E2 -612.312} C_VEL
LIN {X 0,Y 601.411,Z 81.886,A -85,B 0,C 180,E1 -614.409,E2 -614.409} C_VEL
LIN {X 0,Y 601.416,Z 81.877,A -85,B 0,C 180,E1 -617.172,E2 -617.172} C_VEL
LIN {X 0,Y 601.436,Z 81.879,A -85,B 0,C 180,E1 -619.905,E2 -619.905} C_VEL
LIN {X 0,Y 601.44,Z 81.877,A -85,B 0,C 180,E1 -622.615,E2 -622.615} C_VEL
LIN {X 0,Y 601.417,Z 81.877,A -85,B 0,C 180,E1 -625.308,E2 -625.308} C_VEL
LIN {X 0,Y 601.433,Z 81.883,A -85,B 0,C 180,E1 -627.991,E2 -627.991} C_VEL
LIN {X 0,Y 601.448,Z 81.874,A -85,B 0,C 180,E1 -630.67,E2 -630.67} C_VEL
LIN {X 0,Y 601.425,Z 81.877,A -85,B 0,C 180,E1 -633.35,E2 -633.35} C_VEL
LIN {X 0,Y 601.416,Z 81.886,A -85,B 0,C 180,E1 -636.037,E2 -636.037} C_VEL
LIN {X 0,Y 601.413,Z 81.877,A -85,B 0,C 180,E1 -638.738,E2 -638.738} C_VEL
LIN {X 0,Y 601.423,Z 81.879,A -85,B 0,C 180,E1 -641.459,E2 -641.459} C_VEL
LIN {X 0,Y 601.421,Z 81.88,A -85,B 0,C 180,E1 -644.206,E2 -644.206} C_VEL
LIN {X 0,Y 601.431,Z 81.875,A -85,B 0,C 180,E1 -646.986,E2 -646.986} C_VEL
LIN {X 0,Y 601.402,Z 81.887,A -85,B 0,C 180,E1 -649.81,E2 -649.81} C_VEL
LIN {X 0,Y 601.418,Z 81.876,A -85,B 0,C 180,E1 -652.606,E2 -652.606} C_VEL
LIN {X 0,Y 601.4,Z 81.879,A -85,B 0,C 180,E1 -654.879,E2 -654.879} C_VEL
LIN {X 0,Y 601.411,Z 81.884,A -85,B 0,C 180,E1 -657.362,E2 -657.362} C_VEL
LIN {X 0,Y 601.43,Z 81.876,A -85,B 0,C 180,E1 -660.164,E2 -660.164} C_VEL
LIN {X 0,Y 601.425,Z 81.876,A -85,B 0,C 180,E1 -662.716,E2 -662.716} C_VEL
LIN {X 0,Y 601.395,Z 81.884,A -85,B 0,C 180,E1 -665.112,E2 -665.112} C_VEL
LIN {X 0,Y 601.436,Z 81.885,A -85,B 0,C 180,E1 -667.419,E2 -667.419} C_VEL
LIN {X 0,Y 601.403,Z 81.88,A -85,B 0,C 180,E1 -669.996,E2 -669.996} C_VEL
LIN {X 0,Y 601.415,Z 81.878,A -85,B 0,C 180,E1 -672.67,E2 -672.67} C_VEL
LIN {X 0,Y 601.401,Z 81.885,A -85,B 0,C 180,E1 -675.48,E2 -675.48} C_VEL
LIN {X 0,Y 601.422,Z 81.876,A -85,B 0,C 180,E1 -678.408,E2 -678.408} C_VEL
LIN {X 0,Y 601.416,Z 81.882,A -85,B 0,C 180,E1 -680.874,E2 -680.874} C_VEL
LIN {X 0,Y 601.408,Z 81.883,A -85,B 0,C 180,E1 -683.417,E2 -683.417} C_VEL
LIN {X 0,Y 601.435,Z 81.874,A -85,B 0,C 180,E1 -686.065,E2 -686.065} C_VEL
LIN {X 0,Y 601.421,Z 81.879,A -85,B 0,C 180,E1 -688.546,E2 -688.546} C_VEL
LIN {X 0,Y 601.428,Z 81.88,A -85,B 0,C 180,E1 -691.373,E2 -691.373} C_VEL
LIN {X 0,Y 601.4,Z 81.88,A -85,B 0,C 180,E1 -693.636,E2 -693.636} C_VEL
LIN {X 0,Y 601.462,Z 81.872,A -85,B 0,C 180,E1 -695.86,E2 -695.86} C_VEL
LIN {X 0,Y 601.424,Z 81.88,A -85,B 0,C 180,E1 -697.512,E2 -697.512} C_VEL
LIN {X 0,Y 602.334,Z 84.884,A -85,B 0,C 180,E1 -697.588,E2 -697.588} C_VEL
LIN {X 0,Y 602.132,Z 284.852,A -85,B 0,C 180,E1 -700.104,E2 -700.104} C_VEL
LIN {X 0,Y 602.083,Z 301.206,A -85,B 0,C 180,E1 -700.436,E2 -700.436} C_VEL
LIN {X 0,Y 602.015,Z 317.924,A -85,B 0,C 180,E1 -700.921,E2 -700.921} C_VEL
LIN {X 0,Y 601.916,Z 333.534,A -85,B 0,C 180,E1 -701.51,E2 -701.51} C_VEL
LIN {X 0,Y 601.842,Z 348.84,A -85,B 0,C 180,E1 -702.237,E2 -702.237} C_VEL
LIN {X 0,Y 601.765,Z 363.587,A -85,B 0,C 180,E1 -703.089,E2 -703.089} C_VEL
LIN {X 0,Y 601.671,Z 377.775,A -85,B 0,C 180,E1 -704.068,E2 -704.068} C_VEL
LIN {X 0,Y 601.603,Z 390.562,A -85,B 0,C 180,E1 -705.107,E2 -705.107} C_VEL
LIN {X 0,Y 601.526,Z 402.271,A -85,B 0,C 180,E1 -706.214,E2 -706.214} C_VEL
LIN {X 0,Y 601.468,Z 413.966,A -85,B 0,C 180,E1 -707.516,E2 -707.516} C_VEL
LIN {X 0,Y 601.433,Z 424.045,A -85,B 0,C 180,E1 -708.84,E2 -708.84} C_VEL
LIN {X 0,Y 601.389,Z 433.014,A -85,B 0,C 180,E1 -710.244,E2 -710.244} C_VEL
LIN {X 0,Y 601.365,Z 440.277,A -85,B 0,C 180,E1 -711.6,E2 -711.6} C_VEL
LIN {X 0,Y 601.369,Z 446.287,A -85,B 0,C 180,E1 -712.951,E2 -712.951} C_VEL
LIN {X 0,Y 601.352,Z 451.044,A -85,B 0,C 180,E1 -714.299,E2 -714.299} C_VEL
LIN {X 0,Y 601.339,Z 455.539,A -85,B 0,C 180,E1 -715.979,E2 -715.979} C_VEL
LIN {X 0,Y 601.317,Z 458.007,A -85,B 0,C 180,E1 -717.32,E2 -717.32} C_VEL
LIN {X 0,Y 601.343,Z 459.45,A -85,B 0,C 180,E1 -718.661,E2 -718.661} C_VEL
LIN {X 0,Y 601.332,Z 459.996,A -85,B 0,C 180,E1 -720,E2 -720} C_VEL
LIN {X 0,Y 601.341,Z 459.513,A -85,B 0,C 180,E1 -721.339,E2 -721.339} C_VEL
LIN {X 0,Y 601.319,Z 458.152,A -85,B 0,C 180,E1 -722.68,E2 -722.68} C_VEL
LIN {X 0,Y 601.338,Z 455.732,A -85,B 0,C 180,E1 -724.021,E2 -724.021} C_VEL
LIN {X 0,Y 601.345,Z 452.375,A -85,B 0,C 180,E1 -725.365,E2 -725.365} C_VEL
LIN {X 0,Y 601.366,Z 446.635,A -85,B 0,C 180,E1 -727.048,E2 -727.048} C_VEL
LIN {X 0,Y 601.365,Z 440.708,A -85,B 0,C 180,E1 -728.4,E2 -728.4} C_VEL
LIN {X 0,Y 601.383,Z 432.538,A -85,B 0,C 180,E1 -729.926,E2 -729.926} C_VEL
LIN {X 0,Y 601.425,Z 423.732,A -85,B 0,C 180,E1 -731.294,E2 -731.294} C_VEL
LIN {X 0,Y 601.473,Z 413.305,A -85,B 0,C 180,E1 -732.655,E2 -732.655} C_VEL
LIN {X 0,Y 601.532,Z 402.125,A -85,B 0,C 180,E1 -733.891,E2 -733.891} C_VEL
LIN {X 0,Y 601.595,Z 389.625,A -85,B 0,C 180,E1 -735.066,E2 -735.066} C_VEL
LIN {X 0,Y 601.696,Z 376.658,A -85,B 0,C 180,E1 -736.105,E2 -736.105} C_VEL
LIN {X 0,Y 601.751,Z 362.574,A -85,B 0,C 180,E1 -737.064,E2 -737.064} C_VEL
LIN {X 0,Y 601.839,Z 348.888,A -85,B 0,C 180,E1 -737.85,E2 -737.85} C_VEL
LIN {X 0,Y 601.941,Z 333.009,A -85,B 0,C 180,E1 -738.603,E2 -738.603} C_VEL
LIN {X 0,Y 602.011,Z 316.666,A -85,B 0,C 180,E1 -739.212,E2 -739.212} C_VEL
LIN {X 0,Y 602.077,Z 300.349,A -85,B 0,C 180,E1 -739.675,E2 -739.675} C_VEL
LIN {X 0,Y 602.12,Z 283.477,A -85,B 0,C 180,E1 -740.007,E2 -740.007} C_VEL
LIN {X 0,Y 602.272,Z 89.182,A -85,B 0,C 180,E1 -742.45,E2 -742.45} C_VEL
LIN {X 0,Y 602.06,Z 84.156,A -85,B 0,C 180,E1 -742.522,E2 -742.522} C_VEL
LIN {X 0,Y 601.353,Z 81.891,A -85,B 0,C 180,E1 -742.59,E2 -742.59} C_VEL
LIN {X 0,Y 601.377,Z 81.89,A -85,B 0,C 180,E1 -744.88,E2 -744.88} C_VEL
LIN {X 0,Y 601.394,Z 81.884,A -85,B 0,C 180,E1 -747.358,E2 -747.358} C_VEL
LIN {X 0,Y 601.373,Z 81.885,A -85,B 0,C 180,E1 -749.395,E2 -749.395} C_VEL
LIN {X 0,Y 601.384,Z 81.882,A -85,B 0,C 180,E1 -751.728,E2 -751.728} C_VEL
LIN {X 0,Y 601.412,Z 81.881,A -85,B 0,C 180,E1 -754.119,E2 -754.119} C_VEL
LIN {X 0,Y 601.431,Z 81.876,A -85,B 0,C 180,E1 -757.381,E2 -757.381} C_VEL
LIN {X 0,Y 601.398,Z 81.884,A -85,B 0,C 180,E1 -759.996,E2 -759.996} C_VEL
LIN {X 0,Y 601.412,Z 81.881,A -85,B 0,C 180,E1 -762.67,E2 -762.67} C_VEL
LIN {X 0,Y 601.4,Z 81.881,A -85,B 0,C 180,E1 -765.479,E2 -765.479} C_VEL
LIN {X 0,Y 601.427,Z 81.882,A -85,B 0,C 180,E1 -768.235,E2 -768.235} C_VEL
LIN {X 0,Y 601.41,Z 81.878,A -85,B 0,C 180,E1 -770.873,E2 -770.873} C_VEL
LIN {X 0,Y 601.398,Z 81.885,A -85,B 0,C 180,E1 -773.416,E2 -773.416} C_VEL
LIN {X 0,Y 601.434,Z 81.879,A -85,B 0,C 180,E1 -776.064,E2 -776.064} C_VEL
LIN {X 0,Y 601.421,Z 81.878,A -85,B 0,C 180,E1 -778.545,E2 -778.545} C_VEL
LIN {X 0,Y 601.432,Z 81.886,A -85,B 0,C 180,E1 -781.373,E2 -781.373} C_VEL
LIN {X 0,Y 601.449,Z 82.018,A -85,B 0,C 180,E1 -781.588,E2 -781.588} C_VEL
LIN {X 0,Y 602.359,Z 85.356,A -85,B 0,C 180,E1 -781.896,E2 -781.896} C_VEL
LIN {X 0,Y 602.177,Z 120.562,A -85,B 0,C 180,E1 -784.601,E2 -784.601} C_VEL
LIN {X 0,Y 601.975,Z 156.013,A -85,B 0,C 180,E1 -787.267,E2 -787.267} C_VEL
LIN {X 0,Y 602.044,Z 158.974,A -85,B 0,C 180,E1 -787.457,E2 -787.457} C_VEL
LIN {X 0,Y 602.317,Z 165.476,A -85,B 0,C 180,E1 -787.55,E2 -787.55} C_VEL
LIN {X 0,Y 602.12,Z 366.403,A -85,B 0,C 180,E1 -790.081,E2 -790.081} C_VEL
LIN {X 0,Y 602.084,Z 382.982,A -85,B 0,C 180,E1 -790.435,E2 -790.435} C_VEL
LIN {X 0,Y 602.012,Z 397.928,A -85,B 0,C 180,E1 -790.876,E2 -790.876} C_VEL
LIN {X 0,Y 601.916,Z 413.232,A -85,B 0,C 180,E1 -791.452,E2 -791.452} C_VEL
LIN {X 0,Y 601.869,Z 428.005,A -85,B 0,C 180,E1 -792.15,E2 -792.15} C_VEL
LIN {X 0,Y 601.755,Z 441.836,A -85,B 0,C 180,E1 -792.936,E2 -792.936} C_VEL
LIN {X 0,Y 601.695,Z 456.044,A -85,B 0,C 180,E1 -793.894,E2 -793.894} C_VEL
LIN {X 0,Y 601.593,Z 469.121,A -85,B 0,C 180,E1 -794.934,E2 -794.934} C_VEL
LIN {X 0,Y 601.553,Z 481.679,A -85,B 0,C 180,E1 -796.108,E2 -796.108} C_VEL
LIN {X 0,Y 601.474,Z 492.907,A -85,B 0,C 180,E1 -797.344,E2 -797.344} C_VEL
LIN {X 0,Y 601.428,Z 503.282,A -85,B 0,C 180,E1 -798.69,E2 -798.69} C_VEL
LIN {X 0,Y 601.387,Z 512.269,A -85,B 0,C 180,E1 -800.074,E2 -800.074} C_VEL
LIN {X 0,Y 601.364,Z 520.484,A -85,B 0,C 180,E1 -801.599,E2 -801.599} C_VEL
LIN {X 0,Y 601.362,Z 526.466,A -85,B 0,C 180,E1 -802.951,E2 -802.951} C_VEL
LIN {X 0,Y 601.349,Z 532.244,A -85,B 0,C 180,E1 -804.635,E2 -804.635} C_VEL
LIN {X 0,Y 601.337,Z 535.632,A -85,B 0,C 180,E1 -805.978,E2 -805.978} C_VEL
LIN {X 0,Y 601.314,Z 538.086,A -85,B 0,C 180,E1 -807.32,E2 -807.32} C_VEL
LIN {X 0,Y 601.345,Z 539.477,A -85,B 0,C 180,E1 -808.66,E2 -808.66} C_VEL
LIN {X 0,Y 601.33,Z 540,A -85,B 0,C 180,E1 -810,E2 -810} C_VEL
LIN {X 0,Y 601.345,Z 539.478,A -85,B 0,C 180,E1 -811.339,E2 -811.339} C_VEL
LIN {X 0,Y 601.314,Z 538.087,A -85,B 0,C 180,E1 -812.679,E2 -812.679} C_VEL
LIN {X 0,Y 601.337,Z 535.634,A -85,B 0,C 180,E1 -814.021,E2 -814.021} C_VEL
LIN {X 0,Y 601.349,Z 532.247,A -85,B 0,C 180,E1 -815.364,E2 -815.364} C_VEL
LIN {X 0,Y 601.364,Z 526.47,A -85,B 0,C 180,E1 -817.048,E2 -817.048} C_VEL
LIN {X 0,Y 601.377,Z 518.86,A -85,B 0,C 180,E1 -818.738,E2 -818.738} C_VEL
LIN {X 0,Y 601.409,Z 510.249,A -85,B 0,C 180,E1 -820.265,E2 -820.265} C_VEL
LIN {X 0,Y 601.428,Z 500.973,A -85,B 0,C 180,E1 -821.629,E2 -821.629} C_VEL
LIN {X 0,Y 601.482,Z 491.427,A -85,B 0,C 180,E1 -822.826,E2 -822.826} C_VEL
LIN {X 0,Y 601.543,Z 480.625,A -85,B 0,C 180,E1 -823.997,E2 -823.997} C_VEL
LIN {X 0,Y 601.603,Z 468.149,A -85,B 0,C 180,E1 -825.152,E2 -825.152} C_VEL
LIN {X 0,Y 601.707,Z 454.891,A -85,B 0,C 180,E1 -826.192,E2 -826.192} C_VEL
LIN {X 0,Y 601.787,Z 440.44,A -85,B 0,C 180,E1 -827.15,E2 -827.15} C_VEL
LIN {X 0,Y 601.863,Z 426.275,A -85,B 0,C 180,E1 -827.937,E2 -827.937} C_VEL
LIN {X 0,Y 601.942,Z 411.919,A -85,B 0,C 180,E1 -828.604,E2 -828.604} C_VEL
LIN {X 0,Y 602.01,Z 395.361,A -85,B 0,C 180,E1 -829.212,E2 -829.212} C_VEL
LIN {X 0,Y 602.091,Z 379.371,A -85,B 0,C 180,E1 -829.652,E2 -829.652} C_VEL
LIN {X 0,Y 602.14,Z 363.469,A -85,B 0,C 180,E1 -829.961,E2 -829.961} C_VEL
LIN {X 0,Y 602.3,Z 161.046,A -85,B 0,C 180,E1 -832.506,E2 -832.506} C_VEL
LIN {X 0,Y 601.951,Z 158.169,A -85,B 0,C 180,E1 -832.573,E2 -832.573} C_VEL
LIN {X 0,Y 602.177,Z 123.002,A -85,B 0,C 180,E1 -835.213,E2 -835.213} C_VEL
LIN {X 0,Y 602.38,Z 86.583,A -85,B 0,C 180,E1 -838.008,E2 -838.008} C_VEL
LIN {X 0,Y 602.085,Z 84.155,A -85,B 0,C 180,E1 -838.212,E2 -838.212} C_VEL
LIN {X 0,Y 601.435,Z 81.882,A -85,B 0,C 180,E1 -838.436,E2 -838.436} C_VEL
LIN {X 0,Y 601.438,Z 81.875,A -85,B 0,C 180,E1 -841.458,E2 -841.458} C_VEL
LIN {X 0,Y 601.427,Z 81.879,A -85,B 0,C 180,E1 -844.118,E2 -844.118} C_VEL
LIN {X 0,Y 601.432,Z 81.875,A -85,B 0,C 180,E1 -847.382,E2 -847.382} C_VEL
LIN {X 0,Y 601.397,Z 81.882,A -85,B 0,C 180,E1 -849.995,E2 -849.995} C_VEL
LIN {X 0,Y 601.411,Z 81.884,A -85,B 0,C 180,E1 -852.67,E2 -852.67} C_VEL
LIN {X 0,Y 601.422,Z 81.876,A -85,B 0,C 180,E1 -855.482,E2 -855.482} C_VEL
LIN {X 0,Y 601.421,Z 81.886,A -85,B 0,C 180,E1 -858.406,E2 -858.406} C_VEL
LIN {X 0,Y 601.435,Z 81.876,A -85,B 0,C 180,E1 -860.876,E2 -860.876} C_VEL
LIN {X 0,Y 601.428,Z 81.877,A -85,B 0,C 180,E1 -863.735,E2 -863.735} C_VEL
LIN {X 0,Y 601.429,Z 81.883,A -85,B 0,C 180,E1 -866.064,E2 -866.064} C_VEL
LIN {X 0,Y 601.426,Z 81.875,A -85,B 0,C 180,E1 -869.059,E2 -869.059} C_VEL
LIN {X 0,Y 601.421,Z 81.876,A -85,B 0,C 180,E1 -871.373,E2 -871.373} C_VEL
LIN {X 0,Y 601.399,Z 81.882,A -85,B 0,C 180,E1 -873.636,E2 -873.636} C_VEL
LIN {X 0,Y 601.417,Z 81.879,A -85,B 0,C 180,E1 -876.59,E2 -876.59} C_VEL
LIN {X 0,Y 601.421,Z 81.878,A -85,B 0,C 180,E1 -879.478,E2 -879.478} C_VEL
LIN {X 0,Y 601.399,Z 81.883,A -85,B 0,C 180,E1 -882.312,E2 -882.312} C_VEL
LIN {X 0,Y 601.416,Z 81.879,A -85,B 0,C 180,E1 -884.409,E2 -884.409} C_VEL
LIN {X 0,Y 601.416,Z 81.878,A -85,B 0,C 180,E1 -887.172,E2 -887.172} C_VEL
LIN {X 0,Y 601.428,Z 81.884,A -85,B 0,C 180,E1 -889.905,E2 -889.905} C_VEL
LIN {X 0,Y 601.437,Z 81.874,A -85,B 0,C 180,E1 -892.615,E2 -892.615} C_VEL
LIN {X 0,Y 601.416,Z 81.88,A -85,B 0,C 180,E1 -895.308,E2 -895.308} C_VEL
LIN {X 0,Y 601.423,Z 81.881,A -85,B 0,C 180,E1 -897.991,E2 -897.991} C_VEL
LIN {X 0,Y 601.446,Z 81.873,A -85,B 0,C 180,E1 -900.67,E2 -900.67} C_VEL
LIN {X 0,Y 601.423,Z 81.882,A -85,B 0,C 180,E1 -903.35,E2 -903.35} C_VEL
LIN {X 0,Y 601.41,Z 81.88,A -85,B 0,C 180,E1 -906.037,E2 -906.037} C_VEL
LIN {X 0,Y 601.411,Z 81.878,A -85,B 0,C 180,E1 -908.738,E2 -908.738} C_VEL
LIN {X 0,Y 601.431,Z 81.885,A -85,B 0,C 180,E1 -911.458,E2 -911.458} C_VEL
LIN {X 0,Y 601.405,Z 81.878,A -85,B 0,C 180,E1 -912.377,E2 -912.377} C_VEL
LIN {X 0,Y 600.74,Z 81.965,A -85,B 0,C 180,E1 -912.936,E2 -912.936} C_VEL
LIN {X 0,Y 597.89,Z 82.32,A -85,B 0,C 180,E1 -913.844,E2 -913.844} C_VEL
LIN {X 0,Y 595.479,Z 82.621,A -85,B 0,C 180,E1 -914.574,E2 -914.574} C_VEL
LIN {X 0,Y 594.442,Z 82.752,A -85,B 0,C 180,E1 -915.138,E2 -915.138} C_VEL
LIN {X 0,Y 594.357,Z 82.759,A -85,B 0,C 180,E1 -915.329,E2 -915.329} C_VEL
LIN {X 0,Y 594.376,Z 82.755,A -85,B 0,C 180,E1 -917.904,E2 -917.904} C_VEL
LIN {X 0,Y 594.372,Z 82.759,A -85,B 0,C 180,E1 -920.916,E2 -920.916} C_VEL
LIN {X 0,Y 594.388,Z 82.755,A -85,B 0,C 180,E1 -923.704,E2 -923.704} C_VEL
LIN {X 0,Y 594.382,Z 82.756,A -85,B 0,C 180,E1 -926.7,E2 -926.7} C_VEL
LIN {X 0,Y 594.377,Z 82.762,A -85,B 0,C 180,E1 -928.999,E2 -928.999} C_VEL
LIN {X 0,Y 594.388,Z 82.754,A -85,B 0,C 180,E1 -931.645,E2 -931.645} C_VEL
LIN {X 0,Y 594.39,Z 82.755,A -85,B 0,C 180,E1 -934.579,E2 -934.579} C_VEL
LIN {X 0,Y 594.384,Z 82.761,A -85,B 0,C 180,E1 -937.087,E2 -937.087} C_VEL
LIN {X 0,Y 594.374,Z 82.754,A -85,B 0,C 180,E1 -939.775,E2 -939.775} C_VEL
LIN {X 0,Y 594.364,Z 82.757,A -85,B 0,C 180,E1 -942.376,E2 -942.376} C_VEL
LIN {X 0,Y 594.361,Z 82.76,A -85,B 0,C 180,E1 -945.192,E2 -945.192} C_VEL
LIN {X 0,Y 594.37,Z 82.754,A -85,B 0,C 180,E1 -947.625,E2 -947.625} C_VEL
LIN {X 0,Y 594.386,Z 82.756,A -85,B 0,C 180,E1 -950.321,E2 -950.321} C_VEL
LIN {X 0,Y 594.381,Z 82.76,A -85,B 0,C 180,E1 -952.914,E2 -952.914} C_VEL
LIN {X 0,Y 594.379,Z 82.754,A -85,B 0,C 180,E1 -955.862,E2 -955.862} C_VEL
LIN {X 0,Y 594.386,Z 82.762,A -85,B 0,C 180,E1 -958.651,E2 -958.651} C_VEL
LIN {X 0,Y 594.382,Z 82.756,A -85,B 0,C 180,E1 -961.042,E2 -961.042} C_VEL
LIN {X 0,Y 594.385,Z 82.755,A -85,B 0,C 180,E1 -963.977,E2 -963.977} C_VEL
LIN {X 0,Y 594.385,Z 82.76,A -85,B 0,C 180,E1 -966.296,E2 -966.296} C_VEL
LIN {X 0,Y 594.404,Z 82.75,A -85,B 0,C 180,E1 -969.225,E2 -969.225} C_VEL
LIN {X 0,Y 594.35,Z 82.762,A -85,B 0,C 180,E1 -972.095,E2 -972.095} C_VEL
LIN {X 0,Y 594.364,Z 82.763,A -85,B 0,C 180,E1 -974.22,E2 -974.22} C_VEL
LIN {X 0,Y 594.381,Z 82.763,A -85,B 0,C 180,E1 -976.322,E2 -976.322} C_VEL
LIN {X 0,Y 594.376,Z 82.754,A -85,B 0,C 180,E1 -979.095,E2 -979.095} C_VEL
LIN {X 0,Y 594.412,Z 82.753,A -85,B 0,C 180,E1 -981.844,E2 -981.844} C_VEL
LIN {X 0,Y 594.392,Z 82.755,A -85,B 0,C 180,E1 -984.573,E2 -984.573} C_VEL
LIN {X 0,Y 594.403,Z 82.75,A -85,B 0,C 180,E1 -987.29,E2 -987.29} C_VEL
LIN {X 0,Y 594.414,Z 82.758,A -85,B 0,C 180,E1 -990,E2 -990} C_VEL
LIN {X 0,Y 594.405,Z 82.751,A -85,B 0,C 180,E1 -992.711,E2 -992.711} C_VEL
LIN {X 0,Y 594.39,Z 82.754,A -85,B 0,C 180,E1 -995.428,E2 -995.428} C_VEL
LIN {X 0,Y 594.414,Z 82.755,A -85,B 0,C 180,E1 -998.157,E2 -998.157} C_VEL
LIN {X 0,Y 594.392,Z 82.752,A -85,B 0,C 180,E1 -1001.075,E2 -1001.075} C_VEL
LIN {X 0,Y 594.381,Z 82.761,A -85,B 0,C 180,E1 -1003.679,E2 -1003.679} C_VEL
LIN {X 0,Y 594.394,Z 82.751,A -85,B 0,C 180,E1 -1006.719,E2 -1006.719} C_VEL
LIN {X 0,Y 594.367,Z 82.759,A -85,B 0,C 180,E1 -1009.335,E2 -1009.335} C_VEL
LIN {X 0,Y 594.367,Z 82.762,A -85,B 0,C 180,E1 -1011.504,E2 -1011.504} C_VEL
LIN {X 0,Y 594.391,Z 82.752,A -85,B 0,C 180,E1 -1014.446,E2 -1014.446} C_VEL
LIN {X 0,Y 594.383,Z 82.753,A -85,B 0,C 180,E1 -1016.7,E2 -1016.7} C_VEL
LIN {X 0,Y 594.384,Z 82.755,A -85,B 0,C 180,E1 -1018.999,E2 -1018.999} C_VEL
LIN {X 0,Y 594.38,Z 82.761,A -85,B 0,C 180,E1 -1021.643,E2 -1021.643} C_VEL
LIN {X 0,Y 594.379,Z 82.753,A -85,B 0,C 180,E1 -1024.58,E2 -1024.58} C_VEL
LIN {X 0,Y 594.39,Z 82.759,A -85,B 0,C 180,E1 -1027.609,E2 -1027.609} C_VEL
LIN {X 0,Y 594.368,Z 82.755,A -85,B 0,C 180,E1 -1030.567,E2 -1030.567} C_VEL
LIN {X 0,Y 594.37,Z 82.765,A -85,B 0,C 180,E1 -1033.3,E2 -1033.3} C_VEL
LIN {X 0,Y 594.362,Z 82.755,A -85,B 0,C 180,E1 -1036.162,E2 -1036.162} C_VEL
LIN {X 0,Y 594.379,Z 82.754,A -85,B 0,C 180,E1 -1038.536,E2 -1038.536} C_VEL
LIN {X 0,Y 594.385,Z 82.76,A -85,B 0,C 180,E1 -1041.296,E2 -1041.296} C_VEL
LIN {X 0,Y 594.364,Z 82.757,A -85,B 0,C 180,E1 -1043.756,E2 -1043.756} C_VEL
LIN {X 0,Y 594.378,Z 82.754,A -85,B 0,C 180,E1 -1046.239,E2 -1046.239} C_VEL
LIN {X 0,Y 594.372,Z 82.759,A -85,B 0,C 180,E1 -1048.65,E2 -1048.65} C_VEL
LIN {X 0,Y 594.385,Z 82.763,A -85,B 0,C 180,E1 -1051.043,E2 -1051.043} C_VEL
LIN {X 0,Y 594.386,Z 82.758,A -85,B 0,C 180,E1 -1053.301,E2 -1053.301} C_VEL
LIN {X 0,Y 594.38,Z 82.757,A -85,B 0,C 180,E1 -1056.296,E2 -1056.296} C_VEL
LIN {X 0,Y 594.366,Z 82.763,A -85,B 0,C 180,E1 -1057.24,E2 -1057.24} C_VEL
LIN {X 0,Y 595.633,Z 86.142,A -85,B 0,C 180,E1 -1057.338,E2 -1057.338} C_VEL
LIN {X 0,Y 595.587,Z 219.008,A -85,B 0,C 180,E1 -1059.027,E2 -1059.027} C_VEL
LIN {X 0,Y 595.451,Z 284.848,A -85,B 0,C 180,E1 -1059.872,E2 -1059.872} C_VEL
LIN {X 0,Y 595.392,Z 302.169,A -85,B 0,C 180,E1 -1060.229,E2 -1060.229} C_VEL
LIN {X 0,Y 595.297,Z 317.948,A -85,B 0,C 180,E1 -1060.697,E2 -1060.697} C_VEL
LIN {X 0,Y 595.152,Z 333.709,A -85,B 0,C 180,E1 -1061.299,E2 -1061.299} C_VEL
LIN {X 0,Y 595.042,Z 348.831,A -85,B 0,C 180,E1 -1062.027,E2 -1062.027} C_VEL
LIN {X 0,Y 594.9,Z 362.551,A -85,B 0,C 180,E1 -1062.822,E2 -1062.822} C_VEL
LIN {X 0,Y 594.765,Z 377.788,A -85,B 0,C 180,E1 -1063.878,E2 -1063.878} C_VEL
LIN {X 0,Y 594.639,Z 390.568,A -85,B 0,C 180,E1 -1064.929,E2 -1064.929} C_VEL
LIN {X 0,Y 594.565,Z 402.574,A -85,B 0,C 180,E1 -1066.081,E2 -1066.081} C_VEL
LIN {X 0,Y 594.462,Z 413.967,A -85,B 0,C 180,E1 -1067.366,E2 -1067.366} C_VEL
LIN {X 0,Y 594.389,Z 424.296,A -85,B 0,C 180,E1 -1068.744,E2 -1068.744} C_VEL
LIN {X 0,Y 594.333,Z 433.018,A -85,B 0,C 180,E1 -1070.127,E2 -1070.127} C_VEL
LIN {X 0,Y 594.296,Z 440.284,A -85,B 0,C 180,E1 -1071.499,E2 -1071.499} C_VEL
LIN {X 0,Y 594.293,Z 446.289,A -85,B 0,C 180,E1 -1072.867,E2 -1072.867} C_VEL
LIN {X 0,Y 594.282,Z 451.047,A -85,B 0,C 180,E1 -1074.231,E2 -1074.231} C_VEL
LIN {X 0,Y 594.252,Z 455.543,A -85,B 0,C 180,E1 -1075.931,E2 -1075.931} C_VEL
LIN {X 0,Y 594.218,Z 458.004,A -85,B 0,C 180,E1 -1077.288,E2 -1077.288} C_VEL
LIN {X 0,Y 594.242,Z 459.455,A -85,B 0,C 180,E1 -1078.645,E2 -1078.645} C_VEL
LIN {X 0,Y 594.232,Z 459.996,A -85,B 0,C 180,E1 -1080,E2 -1080} C_VEL
LIN {X 0,Y 594.24,Z 459.517,A -85,B 0,C 180,E1 -1081.355,E2 -1081.355} C_VEL
LIN {X 0,Y 594.22,Z 458.149,A -85,B 0,C 180,E1 -1082.712,E2 -1082.712} C_VEL
LIN {X 0,Y 594.251,Z 455.734,A -85,B 0,C 180,E1 -1084.069,E2 -1084.069} C_VEL
LIN {X 0,Y 594.263,Z 452.366,A -85,B 0,C 180,E1 -1085.429,E2 -1085.429} C_VEL
LIN {X 0,Y 594.289,Z 446.628,A -85,B 0,C 180,E1 -1087.133,E2 -1087.133} C_VEL
LIN {X 0,Y 594.296,Z 440.71,A -85,B 0,C 180,E1 -1088.501,E2 -1088.501} C_VEL
LIN {X 0,Y 594.33,Z 432.534,A -85,B 0,C 180,E1 -1090.045,E2 -1090.045} C_VEL
LIN {X 0,Y 594.374,Z 423.87,A -85,B 0,C 180,E1 -1091.409,E2 -1091.409} C_VEL
LIN {X 0,Y 594.447,Z 413.301,A -85,B 0,C 180,E1 -1092.807,E2 -1092.807} C_VEL
LIN {X 0,Y 594.532,Z 401.768,A -85,B 0,C 180,E1 -1094.093,E2 -1094.093} C_VEL
LIN {X 0,Y 594.644,Z 389.608,A -85,B 0,C 180,E1 -1095.246,E2 -1095.246} C_VEL
LIN {X 0,Y 594.801,Z 376.657,A -85,B 0,C 180,E1 -1096.297,E2 -1096.297} C_VEL
LIN {X 0,Y 594.889,Z 362.57,A -85,B 0,C 180,E1 -1097.267,E2 -1097.267} C_VEL
LIN {X 0,Y 595.023,Z 348.859,A -85,B 0,C 180,E1 -1098.062,E2 -1098.062} C_VEL
LIN {X 0,Y 595.186,Z 333.383,A -85,B 0,C 180,E1 -1098.805,E2 -1098.805} C_VEL
LIN {X 0,Y 595.268,Z 317.956,A -85,B 0,C 180,E1 -1099.393,E2 -1099.393} C_VEL
LIN {X 0,Y 595.388,Z 301.266,A -85,B 0,C 180,E1 -1099.883,E2 -1099.883} C_VEL
LIN {X 0,Y 595.445,Z 284.851,A -85,B 0,C 180,E1 -1100.219,E2 -1100.219} C_VEL
LIN {X 0,Y 595.734,Z 91.338,A -85,B 0,C 180,E1 -1102.682,E2 -1102.682} C_VEL
LIN {X 0,Y 595.598,Z 86.243,A -85,B 0,C 180,E1 -1102.752,E2 -1102.752} C_VEL
LIN {X 0,Y 594.304,Z 82.771,A -85,B 0,C 180,E1 -1102.869,E2 -1102.869} C_VEL
LIN {X 0,Y 594.313,Z 82.771,A -85,B 0,C 180,E1 -1105.196,E2 -1105.196} C_VEL
LIN {X 0,Y 594.344,Z 82.761,A -85,B 0,C 180,E1 -1107.518,E2 -1107.518} C_VEL
LIN {X 0,Y 594.331,Z 82.761,A -85,B 0,C 180,E1 -1109.779,E2 -1109.779} C_VEL
LIN {X 0,Y 594.353,Z 82.76,A -85,B 0,C 180,E1 -1112.148,E2 -1112.148} C_VEL
LIN {X 0,Y 594.377,Z 82.764,A -85,B 0,C 180,E1 -1114.58,E2 -1114.58} C_VEL
LIN {X 0,Y 594.384,Z 82.754,A -85,B 0,C 180,E1 -1117.607,E2 -1117.607} C_VEL
LIN {X 0,Y 594.364,Z 82.762,A -85,B 0,C 180,E1 -1120.567,E2 -1120.567} C_VEL
LIN {X 0,Y 594.353,Z 82.758,A -85,B 0,C 180,E1 -1123.301,E2 -1123.301} C_VEL
LIN {X 0,Y 594.377,Z 82.763,A -85,B 0,C 180,E1 -1126.159,E2 -1126.159} C_VEL
LIN {X 0,Y 594.377,Z 82.755,A -85,B 0,C 180,E1 -1129.178,E2 -1129.178} C_VEL
LIN {X 0,Y 594.388,Z 82.759,A -85,B 0,C 180,E1 -1132.059,E2 -1132.059} C_VEL
LIN {X 0,Y 594.352,Z 82.758,A -85,B 0,C 180,E1 -1134.676,E2 -1134.676} C_VEL
LIN {X 0,Y 594.381,Z 82.758,A -85,B 0,C 180,E1 -1137.088,E2 -1137.088} C_VEL
LIN {X 0,Y 594.385,Z 82.761,A -85,B 0,C 180,E1 -1139.672,E2 -1139.672} C_VEL
LIN {X 0,Y 594.4,Z 82.842,A -85,B 0,C 180,E1 -1141.302,E2 -1141.302} C_VEL
LIN {X 0,Y 595.818,Z 87.784,A -85,B 0,C 180,E1 -1141.751,E2 -1141.751} C_VEL
LIN {X 0,Y 595.502,Z 125.417,A -85,B 0,C 180,E1 -1144.671,E2 -1144.671} C_VEL
LIN {X 0,Y 595.223,Z 158.383,A -85,B 0,C 180,E1 -1147.173,E2 -1147.173} C_VEL
LIN {X 0,Y 595.784,Z 163.049,A -85,B 0,C 180,E1 -1147.259,E2 -1147.259} C_VEL
LIN {X 0,Y 595.46,Z 364.909,A -85,B 0,C 180,E1 -1149.826,E2 -1149.826} C_VEL
LIN {X 0,Y 595.408,Z 381.158,A -85,B 0,C 180,E1 -1150.162,E2 -1150.162} C_VEL
LIN {X 0,Y 595.272,Z 397.931,A -85,B 0,C 180,E1 -1150.651,E2 -1150.651} C_VEL
LIN {X 0,Y 595.155,Z 413.474,A -85,B 0,C 180,E1 -1151.245,E2 -1151.245} C_VEL
LIN {X 0,Y 595.056,Z 428.009,A -85,B 0,C 180,E1 -1151.939,E2 -1151.939} C_VEL
LIN {X 0,Y 594.895,Z 441.84,A -85,B 0,C 180,E1 -1152.733,E2 -1152.733} C_VEL
LIN {X 0,Y 594.801,Z 456.047,A -85,B 0,C 180,E1 -1153.702,E2 -1153.702} C_VEL
LIN {X 0,Y 594.648,Z 469.119,A -85,B 0,C 180,E1 -1154.753,E2 -1154.753} C_VEL
LIN {X 0,Y 594.559,Z 481.312,A -85,B 0,C 180,E1 -1155.903,E2 -1155.903} C_VEL
LIN {X 0,Y 594.451,Z 492.906,A -85,B 0,C 180,E1 -1157.192,E2 -1157.192} C_VEL
LIN {X 0,Y 594.382,Z 503.418,A -85,B 0,C 180,E1 -1158.573,E2 -1158.573} C_VEL
LIN {X 0,Y 594.332,Z 512.271,A -85,B 0,C 180,E1 -1159.955,E2 -1159.955} C_VEL
LIN {X 0,Y 594.295,Z 520.485,A -85,B 0,C 180,E1 -1161.499,E2 -1161.499} C_VEL
LIN {X 0,Y 594.284,Z 526.466,A -85,B 0,C 180,E1 -1162.867,E2 -1162.867} C_VEL
LIN {X 0,Y 594.266,Z 532.245,A -85,B 0,C 180,E1 -1164.571,E2 -1164.571} C_VEL
LIN {X 0,Y 594.25,Z 535.633,A -85,B 0,C 180,E1 -1165.93,E2 -1165.93} C_VEL
LIN {X 0,Y 594.215,Z 538.086,A -85,B 0,C 180,E1 -1167.288,E2 -1167.288} C_VEL
LIN {X 0,Y 594.244,Z 539.478,A -85,B 0,C 180,E1 -1168.644,E2 -1168.644} C_VEL
LIN {X 0,Y 594.231,Z 540,A -85,B 0,C 180,E1 -1170,E2 -1170} C_VEL
LIN {X 0,Y 594.244,Z 539.478,A -85,B 0,C 180,E1 -1171.355,E2 -1171.355} C_VEL
LIN {X 0,Y 594.215,Z 538.088,A -85,B 0,C 180,E1 -1172.711,E2 -1172.711} C_VEL
LIN {X 0,Y 594.25,Z 535.635,A -85,B 0,C 180,E1 -1174.069,E2 -1174.069} C_VEL
LIN {X 0,Y 594.282,Z 531.187,A -85,B 0,C 180,E1 -1175.769,E2 -1175.769} C_VEL
LIN {X 0,Y 594.288,Z 526.47,A -85,B 0,C 180,E1 -1177.132,E2 -1177.132} C_VEL
LIN {X 0,Y 594.318,Z 518.86,A -85,B 0,C 180,E1 -1178.843,E2 -1178.843} C_VEL
LIN {X 0,Y 594.359,Z 510.25,A -85,B 0,C 180,E1 -1180.388,E2 -1180.388} C_VEL
LIN {X 0,Y 594.405,Z 500.974,A -85,B 0,C 180,E1 -1181.768,E2 -1181.768} C_VEL
LIN {X 0,Y 594.47,Z 491.428,A -85,B 0,C 180,E1 -1182.98,E2 -1182.98} C_VEL
LIN {X 0,Y 594.538,Z 479.954,A -85,B 0,C 180,E1 -1184.231,E2 -1184.231} C_VEL
LIN {X 0,Y 594.677,Z 468.149,A -85,B 0,C 180,E1 -1185.333,E2 -1185.333} C_VEL
LIN {X 0,Y 594.809,Z 454.888,A -85,B 0,C 180,E1 -1186.385,E2 -1186.385} C_VEL
LIN {X 0,Y 594.949,Z 440.444,A -85,B 0,C 180,E1 -1187.353,E2 -1187.353} C_VEL
LIN {X 0,Y 595.045,Z 426.278,A -85,B 0,C 180,E1 -1188.15,E2 -1188.15} C_VEL
LIN {X 0,Y 595.199,Z 411.129,A -85,B 0,C 180,E1 -1188.854,E2 -1188.854} C_VEL
LIN {X 0,Y 595.278,Z 395.36,A -85,B 0,C 180,E1 -1189.438,E2 -1189.438} C_VEL
LIN {X 0,Y 595.389,Z 379.373,A -85,B 0,C 180,E1 -1189.883,E2 -1189.883} C_VEL
LIN {X 0,Y 595.466,Z 363.469,A -85,B 0,C 180,E1 -1190.195,E2 -1190.195} C_VEL
LIN {X 0,Y 595.74,Z 161.566,A -85,B 0,C 180,E1 -1192.761,E2 -1192.761} C_VEL
LIN {X 0,Y 595.224,Z 158.169,A -85,B 0,C 180,E1 -1192.843,E2 -1192.843} C_VEL
LIN {X 0,Y 595.475,Z 126.644,A -85,B 0,C 180,E1 -1195.236,E2 -1195.236} C_VEL
LIN {X 0,Y 595.784,Z 90.777,A -85,B 0,C 180,E1 -1198.015,E2 -1198.015} C_VEL
LIN {X 0,Y 595.815,Z 87.797,A -85,B 0,C 180,E1 -1198.248,E2 -1198.248} C_VEL
LIN {X 0,Y 594.409,Z 82.76,A -85,B 0,C 180,E1 -1198.74,E2 -1198.74} C_VEL
LIN {X 0,Y 594.388,Z 82.753,A -85,B 0,C 180,E1 -1201.645,E2 -1201.645} C_VEL
LIN {X 0,Y 594.392,Z 82.762,A -85,B 0,C 180,E1 -1204.578,E2 -1204.578} C_VEL
LIN {X 0,Y 594.384,Z 82.753,A -85,B 0,C 180,E1 -1207.608,E2 -1207.608} C_VEL
LIN {X 0,Y 594.367,Z 82.764,A -85,B 0,C 180,E1 -1210.566,E2 -1210.566} C_VEL
LIN {X 0,Y 594.377,Z 82.754,A -85,B 0,C 180,E1 -1213.298,E2 -1213.298} C_VEL
LIN {X 0,Y 594.363,Z 82.762,A -85,B 0,C 180,E1 -1216.16,E2 -1216.16} C_VEL
LIN {X 0,Y 594.374,Z 82.754,A -85,B 0,C 180,E1 -1219.177,E2 -1219.177} C_VEL
LIN {X 0,Y 594.381,Z 82.759,A -85,B 0,C 180,E1 -1222.059,E2 -1222.059} C_VEL
LIN {X 0,Y 594.381,Z 82.756,A -85,B 0,C 180,E1 -1224.672,E2 -1224.672} C_VEL
LIN {X 0,Y 594.372,Z 82.754,A -85,B 0,C 180,E1 -1227.088,E2 -1227.088} C_VEL
LIN {X 0,Y 594.383,Z 82.755,A -85,B 0,C 180,E1 -1229.671,E2 -1229.671} C_VEL
LIN {X 0,Y 594.387,Z 82.756,A -85,B 0,C 180,E1 -1232.54,E2 -1232.54} C_VEL
LIN {X 0,Y 594.374,Z 82.754,A -85,B 0,C 180,E1 -1234.807,E2 -1234.807} C_VEL
LIN {X 0,Y 594.36,Z 82.756,A -85,B 0,C 180,E1 -1237.264,E2 -1237.264} C_VEL
LIN {X 0,Y 594.371,Z 82.764,A -85,B 0,C 180,E1 -1239.946,E2 -1239.946} C_VEL
LIN {X 0,Y 594.387,Z 82.752,A -85,B 0,C 180,E1 -1242.807,E2 -1242.807} C_VEL
LIN {X 0,Y 594.385,Z 82.762,A -85,B 0,C 180,E1 -1245.826,E2 -1245.826} C_VEL
LIN {X 0,Y 594.391,Z 82.754,A -85,B 0,C 180,E1 -1248.404,E2 -1248.404} C_VEL
LIN {X 0,Y 594.378,Z 82.755,A -85,B 0,C 180,E1 -1251.158,E2 -1251.158} C_VEL
LIN {X 0,Y 594.362,Z 82.763,A -85,B 0,C 180,E1 -1253.891,E2 -1253.891} C_VEL
LIN {X 0,Y 594.378,Z 82.753,A -85,B 0,C 180,E1 -1256.611,E2 -1256.611} C_VEL
LIN {X 0,Y 594.416,Z 82.754,A -85,B 0,C 180,E1 -1259.323,E2 -1259.323} C_VEL
LIN {X 0,Y 594.394,Z 82.755,A -85,B 0,C 180,E1 -1262.033,E2 -1262.033} C_VEL
LIN {X 0,Y 594.39,Z 82.752,A -85,B 0,C 180,E1 -1264.748,E2 -1264.748} C_VEL
LIN {X 0,Y 594.389,Z 82.762,A -85,B 0,C 180,E1 -1267.473,E2 -1267.473} C_VEL
LIN {X 0,Y 594.389,Z 82.752,A -85,B 0,C 180,E1 -1270.216,E2 -1270.216} C_VEL
LIN {X 0,Y 594.364,Z 82.759,A -85,B 0,C 180,E1 -1272.983,E2 -1272.983} C_VEL
LIN {X 0,Y 594.357,Z 82.759,A -85,B 0,C 180,E1 -1275.329,E2 -1275.329} C_VEL
LIN {X 0,Y 593.687,Z 82.842,A -85,B 0,C 180,E1 -1275.895,E2 -1275.895} C_VEL
LIN {X 0,Y 590.834,Z 83.197,A -85,B 0,C 180,E1 -1276.813,E2 -1276.813} C_VEL
LIN {X 0,Y 588.429,Z 83.501,A -85,B 0,C 180,E1 -1277.552,E2 -1277.552} C_VEL
LIN {X 0,Y 587.4,Z 83.623,A -85,B 0,C 180,E1 -1278.122,E2 -1278.122} C_VEL
LIN {X 0,Y 587.319,Z 83.633,A -85,B 0,C 180,E1 -1278.315,E2 -1278.315} C_VEL
LIN {X 0,Y 587.326,Z 83.638,A -85,B 0,C 180,E1 -1281.038,E2 -1281.038} C_VEL
LIN {X 0,Y 587.319,Z 83.643,A -85,B 0,C 180,E1 -1283.259,E2 -1283.259} C_VEL
LIN {X 0,Y 587.331,Z 83.636,A -85,B 0,C 180,E1 -1285.517,E2 -1285.517} C_VEL
LIN {X 0,Y 587.344,Z 83.631,A -85,B 0,C 180,E1 -1287.818,E2 -1287.818} C_VEL
LIN {X 0,Y 587.339,Z 83.632,A -85,B 0,C 180,E1 -1290.511,E2 -1290.511} C_VEL
LIN {X 0,Y 587.331,Z 83.636,A -85,B 0,C 180,E1 -1293.397,E2 -1293.397} C_VEL
LIN {X 0,Y 587.353,Z 83.628,A -85,B 0,C 180,E1 -1295.896,E2 -1295.896} C_VEL
LIN {X 0,Y 587.331,Z 83.634,A -85,B 0,C 180,E1 -1298.479,E2 -1298.479} C_VEL
LIN {X 0,Y 587.334,Z 83.637,A -85,B 0,C 180,E1 -1301.157,E2 -1301.157} C_VEL
LIN {X 0,Y 587.323,Z 83.633,A -85,B 0,C 180,E1 -1304.114,E2 -1304.114} C_VEL
LIN {X 0,Y 587.321,Z 83.639,A -85,B 0,C 180,E1 -1306.995,E2 -1306.995} C_VEL
LIN {X 0,Y 587.315,Z 83.633,A -85,B 0,C 180,E1 -1309.746,E2 -1309.746} C_VEL
LIN {X 0,Y 587.342,Z 83.635,A -85,B 0,C 180,E1 -1312.393,E2 -1312.393} C_VEL
LIN {X 0,Y 587.359,Z 83.628,A -85,B 0,C 180,E1 -1315.78,E2 -1315.78} C_VEL
LIN {X 0,Y 587.352,Z 83.633,A -85,B 0,C 180,E1 -1318.232,E2 -1318.232} C_VEL
LIN {X 0,Y 587.348,Z 83.634,A -85,B 0,C 180,E1 -1320.867,E2 -1320.867} C_VEL
LIN {X 0,Y 587.358,Z 83.629,A -85,B 0,C 180,E1 -1323.819,E2 -1323.819} C_VEL
LIN {X 0,Y 587.333,Z 83.634,A -85,B 0,C 180,E1 -1325.994,E2 -1325.994} C_VEL
LIN {X 0,Y 587.322,Z 83.639,A -85,B 0,C 180,E1 -1328.226,E2 -1328.226} C_VEL
LIN {X 0,Y 587.349,Z 83.629,A -85,B 0,C 180,E1 -1331.152,E2 -1331.152} C_VEL
LIN {X 0,Y 587.322,Z 83.637,A -85,B 0,C 180,E1 -1334.025,E2 -1334.025} C_VEL
LIN {X 0,Y 587.358,Z 83.635,A -85,B 0,C 180,E1 -1336.155,E2 -1336.155} C_VEL
LIN {X 0,Y 587.342,Z 83.631,A -85,B 0,C 180,E1 -1338.963,E2 -1338.963} C_VEL
LIN {X 0,Y 587.364,Z 83.63,A -85,B 0,C 180,E1 -1341.745,E2 -1341.745} C_VEL
LIN {X 0,Y 587.357,Z 83.632,A -85,B 0,C 180,E1 -1344.508,E2 -1344.508} C_VEL
LIN {X 0,Y 587.37,Z 83.626,A -85,B 0,C 180,E1 -1347.257,E2 -1347.257} C_VEL
LIN {X 0,Y 587.384,Z 83.634,A -85,B 0,C 180,E1 -1350,E2 -1350} C_VEL
LIN {X 0,Y 587.371,Z 83.627,A -85,B 0,C 180,E1 -1352.744,E2 -1352.744} C_VEL
LIN {X 0,Y 587.356,Z 83.631,A -85,B 0,C 180,E1 -1355.493,E2 -1355.493} C_VEL
LIN {X 0,Y 587.366,Z 83.631,A -85,B 0,C 180,E1 -1358.256,E2 -1358.256} C_VEL
LIN {X 0,Y 587.35,Z 83.629,A -85,B 0,C 180,E1 -1361.134,E2 -1361.134} C_VEL
LIN {X 0,Y 587.367,Z 83.63,A -85,B 0,C 180,E1 -1364.261,E2 -1364.261} C_VEL
LIN {X 0,Y 587.35,Z 83.633,A -85,B 0,C 180,E1 -1367.406,E2 -1367.406} C_VEL
LIN {X 0,Y 587.329,Z 83.633,A -85,B 0,C 180,E1 -1370.305,E2 -1370.305} C_VEL
LIN {X 0,Y 587.323,Z 83.636,A -85,B 0,C 180,E1 -1373.259,E2 -1373.259} C_VEL
LIN {X 0,Y 587.337,Z 83.639,A -85,B 0,C 180,E1 -1375.517,E2 -1375.517} C_VEL
LIN {X 0,Y 587.342,Z 83.636,A -85,B 0,C 180,E1 -1377.818,E2 -1377.818} C_VEL
LIN {X 0,Y 587.337,Z 83.63,A -85,B 0,C 180,E1 -1380.51,E2 -1380.51} C_VEL
LIN {X 0,Y 587.338,Z 83.639,A -85,B 0,C 180,E1 -1383.397,E2 -1383.397} C_VEL
LIN {X 0,Y 587.293,Z 83.639,A -85,B 0,C 180,E1 -1385.9,E2 -1385.9} C_VEL
LIN {X 0,Y 587.324,Z 83.632,A -85,B 0,C 180,E1 -1388.48,E2 -1388.48} C_VEL
LIN {X 0,Y 587.338,Z 83.637,A -85,B 0,C 180,E1 -1391.157,E2 -1391.157} C_VEL
LIN {X 0,Y 587.33,Z 83.632,A -85,B 0,C 180,E1 -1394.114,E2 -1394.114} C_VEL
LIN {X 0,Y 587.314,Z 83.639,A -85,B 0,C 180,E1 -1396.994,E2 -1396.994} C_VEL
LIN {X 0,Y 587.314,Z 83.635,A -85,B 0,C 180,E1 -1399.746,E2 -1399.746} C_VEL
LIN {X 0,Y 587.346,Z 83.63,A -85,B 0,C 180,E1 -1402.392,E2 -1402.392} C_VEL
LIN {X 0,Y 587.352,Z 83.631,A -85,B 0,C 180,E1 -1405.652,E2 -1405.652} C_VEL
LIN {X 0,Y 587.341,Z 83.631,A -85,B 0,C 180,E1 -1408.231,E2 -1408.231} C_VEL
LIN {X 0,Y 587.352,Z 83.637,A -85,B 0,C 180,E1 -1410.867,E2 -1410.867} C_VEL
LIN {X 0,Y 587.34,Z 83.632,A -85,B 0,C 180,E1 -1413.721,E2 -1413.721} C_VEL
LIN {X 0,Y 587.333,Z 83.634,A -85,B 0,C 180,E1 -1415.993,E2 -1415.993} C_VEL
LIN {X 0,Y 587.336,Z 83.64,A -85,B 0,C 180,E1 -1416.953,E2 -1416.953} C_VEL
LIN {X 0,Y 588.334,Z 86.518,A -85,B 0,C 180,E1 -1417.045,E2 -1417.045} C_VEL
LIN {X 0,Y 589.122,Z 88.358,A -85,B 0,C 180,E1 -1417.101,E2 -1417.101} C_VEL
LIN {X 0,Y 588.94,Z 232.468,A -85,B 0,C 180,E1 -1418.951,E2 -1418.951} C_VEL
LIN {X 0,Y 588.789,Z 284.845,A -85,B 0,C 180,E1 -1419.634,E2 -1419.634} C_VEL
LIN {X 0,Y 588.705,Z 302.22,A -85,B 0,C 180,E1 -1419.995,E2 -1419.995} C_VEL
LIN {X 0,Y 588.562,Z 317.946,A -85,B 0,C 180,E1 -1420.467,E2 -1420.467} C_VEL
LIN {X 0,Y 588.405,Z 333.885,A -85,B 0,C 180,E1 -1421.084,E2 -1421.084} C_VEL
LIN {X 0,Y 588.236,Z 348.823,A -85,B 0,C 180,E1 -1421.812,E2 -1421.812} C_VEL
LIN {X 0,Y 588.047,Z 363.722,A -85,B 0,C 180,E1 -1422.689,E2 -1422.689} C_VEL
LIN {X 0,Y 587.892,Z 377.801,A -85,B 0,C 180,E1 -1423.684,E2 -1423.684} C_VEL
LIN {X 0,Y 587.681,Z 390.564,A -85,B 0,C 180,E1 -1424.746,E2 -1424.746} C_VEL
LIN {X 0,Y 587.57,Z 403.223,A -85,B 0,C 180,E1 -1425.981,E2 -1425.981} C_VEL
LIN {X 0,Y 587.428,Z 413.967,A -85,B 0,C 180,E1 -1427.213,E2 -1427.213} C_VEL
LIN {X 0,Y 587.359,Z 423.142,A -85,B 0,C 180,E1 -1428.439,E2 -1428.439} C_VEL
LIN {X 0,Y 587.289,Z 432.009,A -85,B 0,C 180,E1 -1429.833,E2 -1429.833} C_VEL
LIN {X 0,Y 587.241,Z 440.291,A -85,B 0,C 180,E1 -1431.396,E2 -1431.396} C_VEL
LIN {X 0,Y 587.216,Z 446.289,A -85,B 0,C 180,E1 -1432.781,E2 -1432.781} C_VEL
LIN {X 0,Y 587.189,Z 451.05,A -85,B 0,C 180,E1 -1434.161,E2 -1434.161} C_VEL
LIN {X 0,Y 587.133,Z 453.954,A -85,B 0,C 180,E1 -1435.193,E2 -1435.193} C_VEL
LIN {X 0,Y 587.181,Z 456.896,A -85,B 0,C 180,E1 -1436.569,E2 -1436.569} C_VEL
LIN {X 0,Y 587.128,Z 458.845,A -85,B 0,C 180,E1 -1437.942,E2 -1437.942} C_VEL
LIN {X 0,Y 587.139,Z 459.83,A -85,B 0,C 180,E1 -1439.314,E2 -1439.314} C_VEL
LIN {X 0,Y 587.14,Z 459.859,A -85,B 0,C 180,E1 -1440.686,E2 -1440.686} C_VEL
LIN {X 0,Y 587.128,Z 458.948,A -85,B 0,C 180,E1 -1442.058,E2 -1442.058} C_VEL
LIN {X 0,Y 587.18,Z 457.042,A -85,B 0,C 180,E1 -1443.431,E2 -1443.431} C_VEL
LIN {X 0,Y 587.13,Z 454.186,A -85,B 0,C 180,E1 -1444.806,E2 -1444.806} C_VEL
LIN {X 0,Y 587.161,Z 450.267,A -85,B 0,C 180,E1 -1446.184,E2 -1446.184} C_VEL
LIN {X 0,Y 587.2,Z 445.246,A -85,B 0,C 180,E1 -1447.565,E2 -1447.565} C_VEL
LIN {X 0,Y 587.245,Z 439.062,A -85,B 0,C 180,E1 -1448.95,E2 -1448.95} C_VEL
LIN {X 0,Y 587.28,Z 430.489,A -85,B 0,C 180,E1 -1450.515,E2 -1450.515} C_VEL
LIN {X 0,Y 587.367,Z 421.303,A -85,B 0,C 180,E1 -1451.911,E2 -1451.911} C_VEL
LIN {X 0,Y 587.456,Z 410.322,A -85,B 0,C 180,E1 -1453.314,E2 -1453.314} C_VEL
LIN {X 0,Y 587.593,Z 398.963,A -85,B 0,C 180,E1 -1454.547,E2 -1454.547} C_VEL
LIN {X 0,Y 587.745,Z 385.535,A -85,B 0,C 180,E1 -1455.785,E2 -1455.785} C_VEL
LIN {X 0,Y 587.924,Z 371.779,A -85,B 0,C 180,E1 -1456.851,E2 -1456.851} C_VEL
LIN {X 0,Y 588.119,Z 358.254,A -85,B 0,C 180,E1 -1457.741,E2 -1457.741} C_VEL
LIN {X 0,Y 588.3,Z 343.689,A -85,B 0,C 180,E1 -1458.546,E2 -1458.546} C_VEL
LIN {X 0,Y 588.473,Z 328.537,A -85,B 0,C 180,E1 -1459.226,E2 -1459.226} C_VEL
LIN {X 0,Y 588.612,Z 313.933,A -85,B 0,C 180,E1 -1459.758,E2 -1459.758} C_VEL
LIN {X 0,Y 588.726,Z 296.451,A -85,B 0,C 180,E1 -1460.232,E2 -1460.232} C_VEL
LIN {X 0,Y 588.805,Z 281.873,A -85,B 0,C 180,E1 -1460.502,E2 -1460.502} C_VEL
LIN {X 0,Y 589.177,Z 91.104,A -85,B 0,C 180,E1 -1462.951,E2 -1462.951} C_VEL
LIN {X 0,Y 589.045,Z 88.267,A -85,B 0,C 180,E1 -1462.993,E2 -1462.993} C_VEL
LIN {X 0,Y 587.353,Z 84.119,A -85,B 0,C 180,E1 -1463.117,E2 -1463.117} C_VEL
LIN {X 0,Y 587.294,Z 83.646,A -85,B 0,C 180,E1 -1463.141,E2 -1463.141} C_VEL
LIN {X 0,Y 587.296,Z 83.638,A -85,B 0,C 180,E1 -1466.168,E2 -1466.168} C_VEL
LIN {X 0,Y 587.321,Z 83.64,A -85,B 0,C 180,E1 -1469.128,E2 -1469.128} C_VEL
LIN {X 0,Y 587.315,Z 83.635,A -85,B 0,C 180,E1 -1471.83,E2 -1471.83} C_VEL
LIN {X 0,Y 587.338,Z 83.637,A -85,B 0,C 180,E1 -1474.346,E2 -1474.346} C_VEL
LIN {X 0,Y 587.339,Z 83.632,A -85,B 0,C 180,E1 -1477.608,E2 -1477.608} C_VEL
LIN {X 0,Y 587.308,Z 83.644,A -85,B 0,C 180,E1 -1480.255,E2 -1480.255} C_VEL
LIN {X 0,Y 587.306,Z 83.636,A -85,B 0,C 180,E1 -1483.117,E2 -1483.117} C_VEL
LIN {X 0,Y 587.327,Z 83.642,A -85,B 0,C 180,E1 -1486.049,E2 -1486.049} C_VEL
LIN {X 0,Y 587.337,Z 83.632,A -85,B 0,C 180,E1 -1488.925,E2 -1488.925} C_VEL
LIN {X 0,Y 587.33,Z 83.638,A -85,B 0,C 180,E1 -1491.52,E2 -1491.52} C_VEL
LIN {X 0,Y 587.292,Z 83.642,A -85,B 0,C 180,E1 -1494.1,E2 -1494.1} C_VEL
LIN {X 0,Y 587.337,Z 83.634,A -85,B 0,C 180,E1 -1496.603,E2 -1496.603} C_VEL
LIN {X 0,Y 587.336,Z 83.642,A -85,B 0,C 180,E1 -1499.49,E2 -1499.49} C_VEL
LIN {X 0,Y 587.372,Z 83.699,A -85,B 0,C 180,E1 -1501.067,E2 -1501.067} C_VEL
LIN {X 0,Y 589.158,Z 90.468,A -85,B 0,C 180,E1 -1501.661,E2 -1501.661} C_VEL
LIN {X 0,Y 588.962,Z 120.562,A -85,B 0,C 180,E1 -1503.989,E2 -1503.989} C_VEL
LIN {X 0,Y 588.572,Z 154.553,A -85,B 0,C 180,E1 -1506.607,E2 -1506.607} C_VEL
LIN {X 0,Y 588.526,Z 158.436,A -85,B 0,C 180,E1 -1506.903,E2 -1506.903} C_VEL
LIN {X 0,Y 589.235,Z 163.473,A -85,B 0,C 180,E1 -1506.998,E2 -1506.998} C_VEL
LIN {X 0,Y 588.799,Z 366.402,A -85,B 0,C 180,E1 -1509.611,E2 -1509.611} C_VEL
LIN {X 0,Y 588.706,Z 382.986,A -85,B 0,C 180,E1 -1509.972,E2 -1509.972} C_VEL
LIN {X 0,Y 588.533,Z 399.228,A -85,B 0,C 180,E1 -1510.466,E2 -1510.466} C_VEL
LIN {X 0,Y 588.344,Z 415.958,A -85,B 0,C 180,E1 -1511.133,E2 -1511.133} C_VEL
LIN {X 0,Y 588.2,Z 431.296,A -85,B 0,C 180,E1 -1511.901,E2 -1511.901} C_VEL
LIN {X 0,Y 588.032,Z 445.554,A -85,B 0,C 180,E1 -1512.761,E2 -1512.761} C_VEL
LIN {X 0,Y 587.851,Z 459.534,A -85,B 0,C 180,E1 -1513.772,E2 -1513.772} C_VEL
LIN {X 0,Y 587.677,Z 471.067,A -85,B 0,C 180,E1 -1514.746,E2 -1514.746} C_VEL
LIN {X 0,Y 587.558,Z 483.62,A -85,B 0,C 180,E1 -1515.981,E2 -1515.981} C_VEL
LIN {X 0,Y 587.429,Z 494.33,A -85,B 0,C 180,E1 -1517.212,E2 -1517.212} C_VEL
LIN {X 0,Y 587.352,Z 504.673,A -85,B 0,C 180,E1 -1518.613,E2 -1518.613} C_VEL
LIN {X 0,Y 587.289,Z 513.283,A -85,B 0,C 180,E1 -1520.007,E2 -1520.007} C_VEL
LIN {X 0,Y 587.239,Z 520.486,A -85,B 0,C 180,E1 -1521.396,E2 -1521.396} C_VEL
LIN {X 0,Y 587.208,Z 526.466,A -85,B 0,C 180,E1 -1522.78,E2 -1522.78} C_VEL
LIN {X 0,Y 587.19,Z 532.245,A -85,B 0,C 180,E1 -1524.505,E2 -1524.505} C_VEL
LIN {X 0,Y 587.166,Z 535.634,A -85,B 0,C 180,E1 -1525.881,E2 -1525.881} C_VEL
LIN {X 0,Y 587.122,Z 538.087,A -85,B 0,C 180,E1 -1527.255,E2 -1527.255} C_VEL
LIN {X 0,Y 587.144,Z 539.478,A -85,B 0,C 180,E1 -1528.628,E2 -1528.628} C_VEL
LIN {X 0,Y 587.132,Z 540,A -85,B 0,C 180,E1 -1530,E2 -1530} C_VEL
LIN {X 0,Y 587.144,Z 539.479,A -85,B 0,C 180,E1 -1531.371,E2 -1531.371} C_VEL
LIN {X 0,Y 587.122,Z 538.088,A -85,B 0,C 180,E1 -1532.744,E2 -1532.744} C_VEL
LIN {X 0,Y 587.166,Z 535.635,A -85,B 0,C 180,E1 -1534.118,E2 -1534.118} C_VEL
LIN {X 0,Y 587.189,Z 531.188,A -85,B 0,C 180,E1 -1535.839,E2 -1535.839} C_VEL
LIN {X 0,Y 587.211,Z 526.47,A -85,B 0,C 180,E1 -1537.219,E2 -1537.219} C_VEL
LIN {X 0,Y 587.246,Z 518.859,A -85,B 0,C 180,E1 -1538.95,E2 -1538.95} C_VEL
LIN {X 0,Y 587.285,Z 510.252,A -85,B 0,C 180,E1 -1540.515,E2 -1540.515} C_VEL
LIN {X 0,Y 587.365,Z 500.975,A -85,B 0,C 180,E1 -1541.911,E2 -1541.911} C_VEL
LIN {X 0,Y 587.45,Z 491.428,A -85,B 0,C 180,E1 -1543.138,E2 -1543.138} C_VEL
LIN {X 0,Y 587.588,Z 479.575,A -85,B 0,C 180,E1 -1544.441,E2 -1544.441} C_VEL
LIN {X 0,Y 587.758,Z 467.103,A -85,B 0,C 180,E1 -1545.607,E2 -1545.607} C_VEL
LIN {X 0,Y 587.909,Z 453.711,A -85,B 0,C 180,E1 -1546.672,E2 -1546.672} C_VEL
LIN {X 0,Y 588.117,Z 439.013,A -85,B 0,C 180,E1 -1547.651,E2 -1547.651} C_VEL
LIN {X 0,Y 588.288,Z 424.532,A -85,B 0,C 180,E1 -1548.456,E2 -1548.456} C_VEL
LIN {X 0,Y 588.436,Z 409.419,A -85,B 0,C 180,E1 -1549.148,E2 -1549.148} C_VEL
LIN {X 0,Y 588.612,Z 393.269,A -85,B 0,C 180,E1 -1549.735,E2 -1549.735} C_VEL
LIN {X 0,Y 588.759,Z 376.624,A -85,B 0,C 180,E1 -1550.184,E2 -1550.184} C_VEL
LIN {X 0,Y 588.805,Z 360.457,A -85,B 0,C 180,E1 -1550.479,E2 -1550.479} C_VEL
LIN {X 0,Y 589.191,Z 162.232,A -85,B 0,C 180,E1 -1553.02,E2 -1553.02} C_VEL
LIN {X 0,Y 588.518,Z 158.27,A -85,B 0,C 180,E1 -1553.11,E2 -1553.11} C_VEL
LIN {X 0,Y 588.861,Z 126.644,A -85,B 0,C 180,E1 -1555.54,E2 -1555.54} C_VEL
LIN {X 0,Y 589.218,Z 90.771,A -85,B 0,C 180,E1 -1558.334,E2 -1558.334} C_VEL
LIN {X 0,Y 588.054,Z 86.053,A -85,B 0,C 180,E1 -1558.762,E2 -1558.762} C_VEL
LIN {X 0,Y 587.335,Z 83.639,A -85,B 0,C 180,E1 -1559,E2 -1559} C_VEL
LIN {X 0,Y 587.351,Z 83.631,A -85,B 0,C 180,E1 -1561.837,E2 -1561.837} C_VEL
LIN {X 0,Y 587.352,Z 83.636,A -85,B 0,C 180,E1 -1564.349,E2 -1564.349} C_VEL
LIN {X 0,Y 587.339,Z 83.631,A -85,B 0,C 180,E1 -1567.607,E2 -1567.607} C_VEL
LIN {X 0,Y 587.309,Z 83.641,A -85,B 0,C 180,E1 -1570.254,E2 -1570.254} C_VEL
LIN {X 0,Y 587.319,Z 83.635,A -85,B 0,C 180,E1 -1573.005,E2 -1573.005} C_VEL
LIN {X 0,Y 587.322,Z 83.635,A -85,B 0,C 180,E1 -1575.886,E2 -1575.886} C_VEL
LIN {X 0,Y 587.333,Z 83.633,A -85,B 0,C 180,E1 -1578.925,E2 -1578.925} C_VEL
LIN {X 0,Y 587.328,Z 83.632,A -85,B 0,C 180,E1 -1581.521,E2 -1581.521} C_VEL
LIN {X 0,Y 587.345,Z 83.636,A -85,B 0,C 180,E1 -1584.455,E2 -1584.455} C_VEL
LIN {X 0,Y 587.334,Z 83.632,A -85,B 0,C 180,E1 -1586.888,E2 -1586.888} C_VEL
LIN {X 0,Y 587.338,Z 83.631,A -85,B 0,C 180,E1 -1589.489,E2 -1589.489} C_VEL
LIN {X 0,Y 587.347,Z 83.636,A -85,B 0,C 180,E1 -1592.307,E2 -1592.307} C_VEL
LIN {X 0,Y 587.333,Z 83.635,A -85,B 0,C 180,E1 -1594.483,E2 -1594.483} C_VEL
LIN {X 0,Y 587.314,Z 83.633,A -85,B 0,C 180,E1 -1597.131,E2 -1597.131} C_VEL
LIN {X 0,Y 587.324,Z 83.637,A -85,B 0,C 180,E1 -1599.695,E2 -1599.695} C_VEL
LIN {X 0,Y 587.355,Z 83.629,A -85,B 0,C 180,E1 -1602.594,E2 -1602.594} C_VEL
LIN {X 0,Y 587.361,Z 83.635,A -85,B 0,C 180,E1 -1605.739,E2 -1605.739} C_VEL
LIN {X 0,Y 587.343,Z 83.63,A -85,B 0,C 180,E1 -1608.866,E2 -1608.866} C_VEL
LIN {X 0,Y 587.362,Z 83.637,A -85,B 0,C 180,E1 -1611.745,E2 -1611.745} C_VEL
LIN {X 0,Y 587.355,Z 83.629,A -85,B 0,C 180,E1 -1614.507,E2 -1614.507} C_VEL
LIN {X 0,Y 587.368,Z 83.63,A -85,B 0,C 180,E1 -1617.257,E2 -1617.257} C_VEL
LIN {X 0,Y 587.38,Z 83.629,A -85,B 0,C 180,E1 -1620,E2 -1620} C_VEL
LIN {X 0,Y 587.372,Z 83.626,A -85,B 0,C 180,E1 -1622.743,E2 -1622.743} C_VEL
LIN {X 0,Y 587.35,Z 83.639,A -85,B 0,C 180,E1 -1625.493,E2 -1625.493} C_VEL
LIN {X 0,Y 587.362,Z 83.628,A -85,B 0,C 180,E1 -1628.255,E2 -1628.255} C_VEL
LIN {X 0,Y 587.344,Z 83.635,A -85,B 0,C 180,E1 -1631.134,E2 -1631.134} C_VEL
LIN {X 0,Y 587.361,Z 83.627,A -85,B 0,C 180,E1 -1634.261,E2 -1634.261} C_VEL
LIN {X 0,Y 587.355,Z 83.637,A -85,B 0,C 180,E1 -1637.406,E2 -1637.406} C_VEL
LIN {X 0,Y 587.319,Z 83.633,A -85,B 0,C 180,E1 -1638.315,E2 -1638.315} C_VEL
LIN {X 0,Y 586.664,Z 83.718,A -85,B 0,C 180,E1 -1638.887,E2 -1638.887} C_VEL
LIN {X 0,Y 583.833,Z 84.08,A -85,B 0,C 180,E1 -1639.815,E2 -1639.815} C_VEL
LIN {X 0,Y 581.424,Z 84.384,A -85,B 0,C 180,E1 -1640.562,E2 -1640.562} C_VEL
LIN {X 0,Y 580.374,Z 84.51,A -85,B 0,C 180,E1 -1641.138,E2 -1641.138} C_VEL
LIN {X 0,Y 580.279,Z 84.519,A -85,B 0,C 180,E1 -1641.334,E2 -1641.334} C_VEL
LIN {X 0,Y 580.298,Z 84.507,A -85,B 0,C 180,E1 -1644.316,E2 -1644.316} C_VEL
LIN {X 0,Y 580.274,Z 84.512,A -85,B 0,C 180,E1 -1646.624,E2 -1646.624} C_VEL
LIN {X 0,Y 580.298,Z 84.514,A -85,B 0,C 180,E1 -1649.31,E2 -1649.31} C_VEL
LIN {X 0,Y 580.298,Z 84.507,A -85,B 0,C 180,E1 -1652.201,E2 -1652.201} C_VEL
LIN {X 0,Y 580.296,Z 84.512,A -85,B 0,C 180,E1 -1654.696,E2 -1654.696} C_VEL
LIN {X 0,Y 580.297,Z 84.513,A -85,B 0,C 180,E1 -1657.268,E2 -1657.268} C_VEL
LIN {X 0,Y 580.294,Z 84.509,A -85,B 0,C 180,E1 -1660.272,E2 -1660.272} C_VEL
LIN {X 0,Y 580.274,Z 84.517,A -85,B 0,C 180,E1 -1662.707,E2 -1662.707} C_VEL
LIN {X 0,Y 580.271,Z 84.511,A -85,B 0,C 180,E1 -1665.609,E2 -1665.609} C_VEL
LIN {X 0,Y 580.311,Z 84.508,A -85,B 0,C 180,E1 -1668.235,E2 -1668.235} C_VEL
LIN {X 0,Y 580.286,Z 84.515,A -85,B 0,C 180,E1 -1670.966,E2 -1670.966} C_VEL
LIN {X 0,Y 580.265,Z 84.511,A -85,B 0,C 180,E1 -1673.597,E2 -1673.597} C_VEL
LIN {X 0,Y 580.314,Z 84.508,A -85,B 0,C 180,E1 -1676.146,E2 -1676.146} C_VEL
LIN {X 0,Y 580.286,Z 84.519,A -85,B 0,C 180,E1 -1678.616,E2 -1678.616} C_VEL
LIN {X 0,Y 580.291,Z 84.511,A -85,B 0,C 180,E1 -1681.024,E2 -1681.024} C_VEL
LIN {X 0,Y 580.29,Z 84.508,A -85,B 0,C 180,E1 -1683.666,E2 -1683.666} C_VEL
LIN {X 0,Y 580.298,Z 84.508,A -85,B 0,C 180,E1 -1685.684,E2 -1685.684} C_VEL
LIN {X 0,Y 580.272,Z 84.513,A -85,B 0,C 180,E1 -1687.948,E2 -1687.948} C_VEL
LIN {X 0,Y 580.318,Z 84.507,A -85,B 0,C 180,E1 -1690.915,E2 -1690.915} C_VEL
LIN {X 0,Y 580.276,Z 84.512,A -85,B 0,C 180,E1 -1693.826,E2 -1693.826} C_VEL
LIN {X 0,Y 580.325,Z 84.509,A -85,B 0,C 180,E1 -1695.984,E2 -1695.984} C_VEL
LIN {X 0,Y 580.305,Z 84.508,A -85,B 0,C 180,E1 -1698.827,E2 -1698.827} C_VEL
LIN {X 0,Y 580.327,Z 84.506,A -85,B 0,C 180,E1 -1701.644,E2 -1701.644} C_VEL
LIN {X 0,Y 580.324,Z 84.509,A -85,B 0,C 180,E1 -1704.441,E2 -1704.441} C_VEL
LIN {X 0,Y 580.337,Z 84.503,A -85,B 0,C 180,E1 -1707.224,E2 -1707.224} C_VEL
LIN {X 0,Y 580.353,Z 84.51,A -85,B 0,C 180,E1 -1710,E2 -1710} C_VEL
LIN {X 0,Y 580.338,Z 84.503,A -85,B 0,C 180,E1 -1712.777,E2 -1712.777} C_VEL
LIN {X 0,Y 580.322,Z 84.508,A -85,B 0,C 180,E1 -1715.56,E2 -1715.56} C_VEL
LIN {X 0,Y 580.329,Z 84.507,A -85,B 0,C 180,E1 -1718.357,E2 -1718.357} C_VEL
LIN {X 0,Y 580.302,Z 84.508,A -85,B 0,C 180,E1 -1721.191,E2 -1721.191} C_VEL
LIN {X 0,Y 580.327,Z 84.51,A -85,B 0,C 180,E1 -1724.017,E2 -1724.017} C_VEL
LIN {X 0,Y 580.314,Z 84.505,A -85,B 0,C 180,E1 -1726.914,E2 -1726.914} C_VEL
LIN {X 0,Y 580.305,Z 84.515,A -85,B 0,C 180,E1 -1729.823,E2 -1729.823} C_VEL
LIN {X 0,Y 580.296,Z 84.508,A -85,B 0,C 180,E1 -1732.803,E2 -1732.803} C_VEL
LIN {X 0,Y 580.309,Z 84.508,A -85,B 0,C 180,E1 -1735.08,E2 -1735.08} C_VEL
LIN {X 0,Y 580.299,Z 84.509,A -85,B 0,C 180,E1 -1738.186,E2 -1738.186} C_VEL
LIN {X 0,Y 580.285,Z 84.509,A -85,B 0,C 180,E1 -1740.695,E2 -1740.695} C_VEL
LIN {X 0,Y 580.307,Z 84.514,A -85,B 0,C 180,E1 -1743.317,E2 -1743.317} C_VEL
LIN {X 0,Y 580.247,Z 84.518,A -85,B 0,C 180,E1 -1745.757,E2 -1745.757} C_VEL
LIN {X 0,Y 580.287,Z 84.509,A -85,B 0,C 180,E1 -1748.147,E2 -1748.147} C_VEL
LIN {X 0,Y 580.299,Z 84.51,A -85,B 0,C 180,E1 -1750.844,E2 -1750.844} C_VEL
LIN {X 0,Y 580.282,Z 84.514,A -85,B 0,C 180,E1 -1753.658,E2 -1753.658} C_VEL
LIN {X 0,Y 580.276,Z 84.511,A -85,B 0,C 180,E1 -1756.61,E2 -1756.61} C_VEL
LIN {X 0,Y 580.299,Z 84.517,A -85,B 0,C 180,E1 -1759.157,E2 -1759.157} C_VEL
LIN {X 0,Y 580.292,Z 84.508,A -85,B 0,C 180,E1 -1761.927,E2 -1761.927} C_VEL
LIN {X 0,Y 580.284,Z 84.511,A -85,B 0,C 180,E1 -1764.455,E2 -1764.455} C_VEL
LIN {X 0,Y 580.292,Z 84.517,A -85,B 0,C 180,E1 -1766.975,E2 -1766.975} C_VEL
LIN {X 0,Y 580.299,Z 84.512,A -85,B 0,C 180,E1 -1769.425,E2 -1769.425} C_VEL
LIN {X 0,Y 580.301,Z 84.509,A -85,B 0,C 180,E1 -1772.142,E2 -1772.142} C_VEL
LIN {X 0,Y 580.325,Z 84.512,A -85,B 0,C 180,E1 -1775.27,E2 -1775.27} C_VEL
LIN {X 0,Y 580.273,Z 84.52,A -85,B 0,C 180,E1 -1776.67,E2 -1776.67} C_VEL
LIN {X 0,Y 582.016,Z 89.087,A -85,B 0,C 180,E1 -1776.814,E2 -1776.814} C_VEL
LIN {X 0,Y 582.659,Z 90.398,A -85,B 0,C 180,E1 -1776.859,E2 -1776.859} C_VEL
LIN {X 0,Y 582.177,Z 275.672,A -85,B 0,C 180,E1 -1779.253,E2 -1779.253} C_VEL
LIN {X 0,Y 582.101,Z 293.337,A -85,B 0,C 180,E1 -1779.551,E2 -1779.551} C_VEL
LIN {X 0,Y 581.965,Z 309.585,A -85,B 0,C 180,E1 -1779.961,E2 -1779.961} C_VEL
LIN {X 0,Y 581.766,Z 325.637,A -85,B 0,C 180,E1 -1780.516,E2 -1780.516} C_VEL
LIN {X 0,Y 581.54,Z 339.958,A -85,B 0,C 180,E1 -1781.139,E2 -1781.139} C_VEL
LIN {X 0,Y 581.32,Z 355.285,A -85,B 0,C 180,E1 -1781.953,E2 -1781.953} C_VEL
LIN {X 0,Y 581.097,Z 368.941,A -85,B 0,C 180,E1 -1782.835,E2 -1782.835} C_VEL
LIN {X 0,Y 580.929,Z 381.179,A -85,B 0,C 180,E1 -1783.754,E2 -1783.754} C_VEL
LIN {X 0,Y 580.719,Z 392.519,A -85,B 0,C 180,E1 -1784.739,E2 -1784.739} C_VEL
LIN {X 0,Y 580.565,Z 404.882,A -85,B 0,C 180,E1 -1785.989,E2 -1785.989} C_VEL
LIN {X 0,Y 580.413,Z 415.329,A -85,B 0,C 180,E1 -1787.233,E2 -1787.233} C_VEL
LIN {X 0,Y 580.323,Z 424.327,A -85,B 0,C 180,E1 -1788.474,E2 -1788.474} C_VEL
LIN {X 0,Y 580.217,Z 433.025,A -85,B 0,C 180,E1 -1789.884,E2 -1789.884} C_VEL
LIN {X 0,Y 580.168,Z 440.298,A -85,B 0,C 180,E1 -1791.291,E2 -1791.291} C_VEL
LIN {X 0,Y 580.126,Z 446.287,A -85,B 0,C 180,E1 -1792.692,E2 -1792.692} C_VEL
LIN {X 0,Y 580.1,Z 451.054,A -85,B 0,C 180,E1 -1794.089,E2 -1794.089} C_VEL
LIN {X 0,Y 580.037,Z 453.96,A -85,B 0,C 180,E1 -1795.135,E2 -1795.135} C_VEL
LIN {X 0,Y 580.107,Z 456.893,A -85,B 0,C 180,E1 -1796.527,E2 -1796.527} C_VEL
LIN {X 0,Y 580.028,Z 458.848,A -85,B 0,C 180,E1 -1797.917,E2 -1797.917} C_VEL
LIN {X 0,Y 580.039,Z 459.824,A -85,B 0,C 180,E1 -1799.306,E2 -1799.306} C_VEL
LIN {X 0,Y 580.04,Z 459.852,A -85,B 0,C 180,E1 -1800.694,E2 -1800.694} C_VEL
LIN {X 0,Y 580.027,Z 458.941,A -85,B 0,C 180,E1 -1802.083,E2 -1802.083} C_VEL
LIN {X 0,Y 580.106,Z 457.038,A -85,B 0,C 180,E1 -1803.473,E2 -1803.473} C_VEL
LIN {X 0,Y 580.034,Z 454.189,A -85,B 0,C 180,E1 -1804.865,E2 -1804.865} C_VEL
LIN {X 0,Y 580.078,Z 450.266,A -85,B 0,C 180,E1 -1806.26,E2 -1806.26} C_VEL
LIN {X 0,Y 580.118,Z 445.247,A -85,B 0,C 180,E1 -1807.658,E2 -1807.658} C_VEL
LIN {X 0,Y 580.156,Z 439.052,A -85,B 0,C 180,E1 -1809.061,E2 -1809.061} C_VEL
LIN {X 0,Y 580.234,Z 431.508,A -85,B 0,C 180,E1 -1810.468,E2 -1810.468} C_VEL
LIN {X 0,Y 580.335,Z 422.543,A -85,B 0,C 180,E1 -1811.881,E2 -1811.881} C_VEL
LIN {X 0,Y 580.428,Z 411.81,A -85,B 0,C 180,E1 -1813.3,E2 -1813.3} C_VEL
LIN {X 0,Y 580.573,Z 401.766,A -85,B 0,C 180,E1 -1814.436,E2 -1814.436} C_VEL
LIN {X 0,Y 580.735,Z 391.54,A -85,B 0,C 180,E1 -1815.441,E2 -1815.441} C_VEL
LIN {X 0,Y 580.965,Z 378.943,A -85,B 0,C 180,E1 -1816.516,E2 -1816.516} C_VEL
LIN {X 0,Y 581.179,Z 365.129,A -85,B 0,C 180,E1 -1817.522,E2 -1817.522} C_VEL
LIN {X 0,Y 581.375,Z 350.453,A -85,B 0,C 180,E1 -1818.41,E2 -1818.41} C_VEL
LIN {X 0,Y 581.636,Z 335.056,A -85,B 0,C 180,E1 -1819.182,E2 -1819.182} C_VEL
LIN {X 0,Y 581.827,Z 319.209,A -85,B 0,C 180,E1 -1819.814,E2 -1819.814} C_VEL
LIN {X 0,Y 582.014,Z 303.801,A -85,B 0,C 180,E1 -1820.291,E2 -1820.291} C_VEL
LIN {X 0,Y 582.138,Z 286.142,A -85,B 0,C 180,E1 -1820.679,E2 -1820.679} C_VEL
LIN {X 0,Y 582.341,Z 216.229,A -85,B 0,C 180,E1 -1821.601,E2 -1821.601} C_VEL
LIN {X 0,Y 582.643,Z 90.961,A -85,B 0,C 180,E1 -1823.224,E2 -1823.224} C_VEL
LIN {X 0,Y 580.229,Z 84.525,A -85,B 0,C 180,E1 -1823.424,E2 -1823.424} C_VEL
LIN {X 0,Y 580.253,Z 84.517,A -85,B 0,C 180,E1 -1826.325,E2 -1826.325} C_VEL
LIN {X 0,Y 580.262,Z 84.517,A -85,B 0,C 180,E1 -1829.302,E2 -1829.302} C_VEL
LIN {X 0,Y 580.286,Z 84.513,A -85,B 0,C 180,E1 -1832.201,E2 -1832.201} C_VEL
LIN {X 0,Y 580.286,Z 84.518,A -85,B 0,C 180,E1 -1834.696,E2 -1834.696} C_VEL
LIN {X 0,Y 580.287,Z 84.511,A -85,B 0,C 180,E1 -1837.269,E2 -1837.269} C_VEL
LIN {X 0,Y 580.287,Z 84.518,A -85,B 0,C 180,E1 -1840.269,E2 -1840.269} C_VEL
LIN {X 0,Y 580.274,Z 84.514,A -85,B 0,C 180,E1 -1842.706,E2 -1842.706} C_VEL
LIN {X 0,Y 580.264,Z 84.516,A -85,B 0,C 180,E1 -1845.609,E2 -1845.609} C_VEL
LIN {X 0,Y 580.282,Z 84.516,A -85,B 0,C 180,E1 -1848.231,E2 -1848.231} C_VEL
LIN {X 0,Y 580.278,Z 84.512,A -85,B 0,C 180,E1 -1850.965,E2 -1850.965} C_VEL
LIN {X 0,Y 580.269,Z 84.52,A -85,B 0,C 180,E1 -1853.596,E2 -1853.596} C_VEL
LIN {X 0,Y 580.317,Z 84.511,A -85,B 0,C 180,E1 -1856.145,E2 -1856.145} C_VEL
LIN {X 0,Y 580.278,Z 84.515,A -85,B 0,C 180,E1 -1858.614,E2 -1858.614} C_VEL
LIN {X 0,Y 580.346,Z 84.664,A -85,B 0,C 180,E1 -1860.833,E2 -1860.833} C_VEL
LIN {X 0,Y 582.438,Z 92.305,A -85,B 0,C 180,E1 -1861.519,E2 -1861.519} C_VEL
LIN {X 0,Y 582.222,Z 129.181,A -85,B 0,C 180,E1 -1864.348,E2 -1864.348} C_VEL
LIN {X 0,Y 581.873,Z 158.728,A -85,B 0,C 180,E1 -1866.627,E2 -1866.627} C_VEL
LIN {X 0,Y 582.723,Z 164.689,A -85,B 0,C 180,E1 -1866.742,E2 -1866.742} C_VEL
LIN {X 0,Y 582.139,Z 366.401,A -85,B 0,C 180,E1 -1869.367,E2 -1869.367} C_VEL
LIN {X 0,Y 582.018,Z 382.987,A -85,B 0,C 180,E1 -1869.732,E2 -1869.732} C_VEL
LIN {X 0,Y 581.835,Z 399.229,A -85,B 0,C 180,E1 -1870.232,E2 -1870.232} C_VEL
LIN {X 0,Y 581.625,Z 414.996,A -85,B 0,C 180,E1 -1870.862,E2 -1870.862} C_VEL
LIN {X 0,Y 581.444,Z 429.711,A -85,B 0,C 180,E1 -1871.592,E2 -1871.592} C_VEL
LIN {X 0,Y 581.205,Z 444.53,A -85,B 0,C 180,E1 -1872.485,E2 -1872.485} C_VEL
LIN {X 0,Y 580.966,Z 458.376,A -85,B 0,C 180,E1 -1873.484,E2 -1873.484} C_VEL
LIN {X 0,Y 580.743,Z 471.066,A -85,B 0,C 180,E1 -1874.559,E2 -1874.559} C_VEL
LIN {X 0,Y 580.59,Z 482.617,A -85,B 0,C 180,E1 -1875.699,E2 -1875.699} C_VEL
LIN {X 0,Y 580.414,Z 494.332,A -85,B 0,C 180,E1 -1877.055,E2 -1877.055} C_VEL
LIN {X 0,Y 580.316,Z 504.673,A -85,B 0,C 180,E1 -1878.473,E2 -1878.473} C_VEL
LIN {X 0,Y 580.218,Z 513.282,A -85,B 0,C 180,E1 -1879.884,E2 -1879.884} C_VEL
LIN {X 0,Y 580.165,Z 520.486,A -85,B 0,C 180,E1 -1881.29,E2 -1881.29} C_VEL
LIN {X 0,Y 580.119,Z 526.465,A -85,B 0,C 180,E1 -1882.691,E2 -1882.691} C_VEL
LIN {X 0,Y 580.114,Z 532.246,A -85,B 0,C 180,E1 -1884.438,E2 -1884.438} C_VEL
LIN {X 0,Y 580.084,Z 535.635,A -85,B 0,C 180,E1 -1885.831,E2 -1885.831} C_VEL
LIN {X 0,Y 580.033,Z 538.088,A -85,B 0,C 180,E1 -1887.222,E2 -1887.222} C_VEL
LIN {X 0,Y 580.044,Z 539.479,A -85,B 0,C 180,E1 -1888.611,E2 -1888.611} C_VEL
LIN {X 0,Y 580.033,Z 540,A -85,B 0,C 180,E1 -1890,E2 -1890} C_VEL
LIN {X 0,Y 580.044,Z 539.479,A -85,B 0,C 180,E1 -1891.388,E2 -1891.388} C_VEL
LIN {X 0,Y 580.033,Z 538.089,A -85,B 0,C 180,E1 -1892.778,E2 -1892.778} C_VEL
LIN {X 0,Y 580.084,Z 535.636,A -85,B 0,C 180,E1 -1894.168,E2 -1894.168} C_VEL
LIN {X 0,Y 580.1,Z 531.189,A -85,B 0,C 180,E1 -1895.91,E2 -1895.91} C_VEL
LIN {X 0,Y 580.121,Z 526.47,A -85,B 0,C 180,E1 -1897.308,E2 -1897.308} C_VEL
LIN {X 0,Y 580.18,Z 518.859,A -85,B 0,C 180,E1 -1899.06,E2 -1899.06} C_VEL
LIN {X 0,Y 580.21,Z 510.253,A -85,B 0,C 180,E1 -1900.644,E2 -1900.644} C_VEL
LIN {X 0,Y 580.334,Z 500.977,A -85,B 0,C 180,E1 -1902.058,E2 -1902.058} C_VEL
LIN {X 0,Y 580.441,Z 491.428,A -85,B 0,C 180,E1 -1903.3,E2 -1903.3} C_VEL
LIN {X 0,Y 580.622,Z 479.936,A -85,B 0,C 180,E1 -1904.581,E2 -1904.581} C_VEL
LIN {X 0,Y 580.813,Z 468.148,A -85,B 0,C 180,E1 -1905.708,E2 -1905.708} C_VEL
LIN {X 0,Y 581.011,Z 454.882,A -85,B 0,C 180,E1 -1906.785,E2 -1906.785} C_VEL
LIN {X 0,Y 581.263,Z 440.436,A -85,B 0,C 180,E1 -1907.775,E2 -1907.775} C_VEL
LIN {X 0,Y 581.478,Z 426.285,A -85,B 0,C 180,E1 -1908.589,E2 -1908.589} C_VEL
LIN {X 0,Y 581.706,Z 411.091,A -85,B 0,C 180,E1 -1909.31,E2 -1909.31} C_VEL
LIN {X 0,Y 581.907,Z 395.358,A -85,B 0,C 180,E1 -1909.903,E2 -1909.903} C_VEL
LIN {X 0,Y 582.036,Z 379.371,A -85,B 0,C 180,E1 -1910.359,E2 -1910.359} C_VEL
LIN {X 0,Y 582.148,Z 363.468,A -85,B 0,C 180,E1 -1910.678,E2 -1910.678} C_VEL
LIN {X 0,Y 582.689,Z 164.963,A -85,B 0,C 180,E1 -1913.256,E2 -1913.256} C_VEL
LIN {X 0,Y 581.867,Z 158.854,A -85,B 0,C 180,E1 -1913.372,E2 -1913.372} C_VEL
LIN {X 0,Y 582.196,Z 130.289,A -85,B 0,C 180,E1 -1915.566,E2 -1915.566} C_VEL
LIN {X 0,Y 582.541,Z 95.616,A -85,B 0,C 180,E1 -1918.274,E2 -1918.274} C_VEL
LIN {X 0,Y 582.503,Z 91.836,A -85,B 0,C 180,E1 -1918.575,E2 -1918.575} C_VEL
LIN {X 0,Y 580.3,Z 84.513,A -85,B 0,C 180,E1 -1919.279,E2 -1919.279} C_VEL
LIN {X 0,Y 580.299,Z 84.513,A -85,B 0,C 180,E1 -1922.2,E2 -1922.2} C_VEL
LIN {X 0,Y 580.292,Z 84.518,A -85,B 0,C 180,E1 -1924.695,E2 -1924.695} C_VEL
LIN {X 0,Y 580.294,Z 84.51,A -85,B 0,C 180,E1 -1927.268,E2 -1927.268} C_VEL
LIN {X 0,Y 580.288,Z 84.516,A -85,B 0,C 180,E1 -1930.27,E2 -1930.27} C_VEL
LIN {X 0,Y 580.279,Z 84.516,A -85,B 0,C 180,E1 -1932.705,E2 -1932.705} C_VEL
LIN {X 0,Y 580.265,Z 84.512,A -85,B 0,C 180,E1 -1935.609,E2 -1935.609} C_VEL
LIN {X 0,Y 580.276,Z 84.518,A -85,B 0,C 180,E1 -1938.231,E2 -1938.231} C_VEL
LIN {X 0,Y 580.286,Z 84.51,A -85,B 0,C 180,E1 -1940.966,E2 -1940.966} C_VEL
LIN {X 0,Y 580.289,Z 84.51,A -85,B 0,C 180,E1 -1943.598,E2 -1943.598} C_VEL
LIN {X 0,Y 580.314,Z 84.514,A -85,B 0,C 180,E1 -1946.145,E2 -1946.145} C_VEL
LIN {X 0,Y 580.282,Z 84.513,A -85,B 0,C 180,E1 -1948.615,E2 -1948.615} C_VEL
LIN {X 0,Y 580.289,Z 84.508,A -85,B 0,C 180,E1 -1951.024,E2 -1951.024} C_VEL
LIN {X 0,Y 580.288,Z 84.512,A -85,B 0,C 180,E1 -1953.665,E2 -1953.665} C_VEL
LIN {X 0,Y 580.297,Z 84.511,A -85,B 0,C 180,E1 -1955.684,E2 -1955.684} C_VEL
LIN {X 0,Y 580.27,Z 84.52,A -85,B 0,C 180,E1 -1957.947,E2 -1957.947} C_VEL
LIN {X 0,Y 580.295,Z 84.508,A -85,B 0,C 180,E1 -1960.913,E2 -1960.913} C_VEL
LIN {X 0,Y 580.306,Z 84.507,A -85,B 0,C 180,E1 -1963.103,E2 -1963.103} C_VEL
LIN {X 0,Y 580.323,Z 84.512,A -85,B 0,C 180,E1 -1965.983,E2 -1965.983} C_VEL
LIN {X 0,Y 580.3,Z 84.507,A -85,B 0,C 180,E1 -1968.827,E2 -1968.827} C_VEL
LIN {X 0,Y 580.325,Z 84.512,A -85,B 0,C 180,E1 -1971.644,E2 -1971.644} C_VEL
LIN {X 0,Y 580.321,Z 84.505,A -85,B 0,C 180,E1 -1974.44,E2 -1974.44} C_VEL
LIN {X 0,Y 580.334,Z 84.506,A -85,B 0,C 180,E1 -1977.224,E2 -1977.224} C_VEL
LIN {X 0,Y 580.349,Z 84.505,A -85,B 0,C 180,E1 -1980,E2 -1980} C_VEL
LIN {X 0,Y 580.338,Z 84.503,A -85,B 0,C 180,E1 -1982.777,E2 -1982.777} C_VEL
LIN {X 0,Y 580.317,Z 84.515,A -85,B 0,C 180,E1 -1985.56,E2 -1985.56} C_VEL
LIN {X 0,Y 580.325,Z 84.504,A -85,B 0,C 180,E1 -1988.356,E2 -1988.356} C_VEL
LIN {X 0,Y 580.296,Z 84.514,A -85,B 0,C 180,E1 -1991.191,E2 -1991.191} C_VEL
LIN {X 0,Y 580.322,Z 84.506,A -85,B 0,C 180,E1 -1994.017,E2 -1994.017} C_VEL
LIN {X 0,Y 580.308,Z 84.51,A -85,B 0,C 180,E1 -1996.914,E2 -1996.914} C_VEL
LIN {X 0,Y 580.301,Z 84.509,A -85,B 0,C 180,E1 -1999.822,E2 -1999.822} C_VEL
LIN {X 0,Y 580.279,Z 84.519,A -85,B 0,C 180,E1 -2001.334,E2 -2001.334} C_VEL
LIN {X 0,Y 579.584,Z 84.599,A -85,B 0,C 180,E1 -2001.913,E2 -2001.913} C_VEL
LIN {X 0,Y 576.708,Z 84.959,A -85,B 0,C 180,E1 -2002.853,E2 -2002.853} C_VEL
LIN {X 0,Y 574.313,Z 85.257,A -85,B 0,C 180,E1 -2003.609,E2 -2003.609} C_VEL
LIN {X 0,Y 573.314,Z 85.378,A -85,B 0,C 180,E1 -2004.193,E2 -2004.193} C_VEL
LIN {X 0,Y 573.247,Z 85.386,A -85,B 0,C 180,E1 -2004.39,E2 -2004.39} C_VEL
LIN {X 0,Y 573.247,Z 85.393,A -85,B 0,C 180,E1 -2006.976,E2 -2006.976} C_VEL
LIN {X 0,Y 573.244,Z 85.39,A -85,B 0,C 180,E1 -2009.489,E2 -2009.489} C_VEL
LIN {X 0,Y 573.25,Z 85.385,A -85,B 0,C 180,E1 -2012.229,E2 -2012.229} C_VEL
LIN {X 0,Y 573.247,Z 85.391,A -85,B 0,C 180,E1 -2014.774,E2 -2014.774} C_VEL
LIN {X 0,Y 573.251,Z 85.392,A -85,B 0,C 180,E1 -2017.167,E2 -2017.167} C_VEL
LIN {X 0,Y 573.246,Z 85.387,A -85,B 0,C 180,E1 -2019.607,E2 -2019.607} C_VEL
LIN {X 0,Y 573.237,Z 85.393,A -85,B 0,C 180,E1 -2022.642,E2 -2022.642} C_VEL
LIN {X 0,Y 573.236,Z 85.387,A -85,B 0,C 180,E1 -2025.667,E2 -2025.667} C_VEL
LIN {X 0,Y 573.242,Z 85.392,A -85,B 0,C 180,E1 -2028.545,E2 -2028.545} C_VEL
LIN {X 0,Y 573.245,Z 85.388,A -85,B 0,C 180,E1 -2031.299,E2 -2031.299} C_VEL
LIN {X 0,Y 573.21,Z 85.391,A -85,B 0,C 180,E1 -2034.019,E2 -2034.019} C_VEL
LIN {X 0,Y 573.283,Z 85.389,A -85,B 0,C 180,E1 -2036.519,E2 -2036.519} C_VEL
LIN {X 0,Y 573.234,Z 85.39,A -85,B 0,C 180,E1 -2039.117,E2 -2039.117} C_VEL
LIN {X 0,Y 573.25,Z 85.387,A -85,B 0,C 180,E1 -2041.971,E2 -2041.971} C_VEL
LIN {X 0,Y 573.254,Z 85.394,A -85,B 0,C 180,E1 -2044.59,E2 -2044.59} C_VEL
LIN {X 0,Y 573.236,Z 85.387,A -85,B 0,C 180,E1 -2047.663,E2 -2047.663} C_VEL
LIN {X 0,Y 573.278,Z 85.386,A -85,B 0,C 180,E1 -2050.729,E2 -2050.729} C_VEL
LIN {X 0,Y 573.249,Z 85.386,A -85,B 0,C 180,E1 -2053.622,E2 -2053.622} C_VEL
LIN {X 0,Y 573.273,Z 85.385,A -85,B 0,C 180,E1 -2055.808,E2 -2055.808} C_VEL
LIN {X 0,Y 573.263,Z 85.386,A -85,B 0,C 180,E1 -2058.745,E2 -2058.745} C_VEL
LIN {X 0,Y 573.283,Z 85.382,A -85,B 0,C 180,E1 -2061.541,E2 -2061.541} C_VEL
LIN {X 0,Y 573.291,Z 85.387,A -85,B 0,C 180,E1 -2064.372,E2 -2064.372} C_VEL
LIN {X 0,Y 573.312,Z 85.384,A -85,B 0,C 180,E1 -2067.893,E2 -2067.893} C_VEL
LIN {X 0,Y 573.332,Z 85.376,A -85,B 0,C 180,E1 -2070.703,E2 -2070.703} C_VEL
LIN {X 0,Y 573.304,Z 85.379,A -85,B 0,C 180,E1 -2072.811,E2 -2072.811} C_VEL
LIN {X 0,Y 573.29,Z 85.385,A -85,B 0,C 180,E1 -2075.629,E2 -2075.629} C_VEL
LIN {X 0,Y 573.285,Z 85.383,A -85,B 0,C 180,E1 -2078.46,E2 -2078.46} C_VEL
LIN {X 0,Y 573.274,Z 85.384,A -85,B 0,C 180,E1 -2081.312,E2 -2081.312} C_VEL
LIN {X 0,Y 573.283,Z 85.383,A -85,B 0,C 180,E1 -2084.425,E2 -2084.425} C_VEL
LIN {X 0,Y 573.26,Z 85.385,A -85,B 0,C 180,E1 -2087.112,E2 -2087.112} C_VEL
LIN {X 0,Y 573.253,Z 85.389,A -85,B 0,C 180,E1 -2090.077,E2 -2090.077} C_VEL
LIN {X 0,Y 573.237,Z 85.389,A -85,B 0,C 180,E1 -2093.1,E2 -2093.1} C_VEL
LIN {X 0,Y 573.257,Z 85.391,A -85,B 0,C 180,E1 -2095.41,E2 -2095.41} C_VEL
LIN {X 0,Y 573.249,Z 85.388,A -85,B 0,C 180,E1 -2098.028,E2 -2098.028} C_VEL
LIN {X 0,Y 573.247,Z 85.387,A -85,B 0,C 180,E1 -2100.176,E2 -2100.176} C_VEL
LIN {X 0,Y 573.257,Z 85.385,A -85,B 0,C 180,E1 -2102.645,E2 -2102.645} C_VEL
LIN {X 0,Y 573.209,Z 85.396,A -85,B 0,C 180,E1 -2105.188,E2 -2105.188} C_VEL
LIN {X 0,Y 573.236,Z 85.391,A -85,B 0,C 180,E1 -2107.808,E2 -2107.808} C_VEL
LIN {X 0,Y 573.247,Z 85.386,A -85,B 0,C 180,E1 -2110.525,E2 -2110.525} C_VEL
LIN {X 0,Y 573.243,Z 85.395,A -85,B 0,C 180,E1 -2113.359,E2 -2113.359} C_VEL
LIN {X 0,Y 573.241,Z 85.386,A -85,B 0,C 180,E1 -2116.332,E2 -2116.332} C_VEL
LIN {X 0,Y 573.231,Z 85.389,A -85,B 0,C 180,E1 -2118.543,E2 -2118.543} C_VEL
LIN {X 0,Y 573.246,Z 85.394,A -85,B 0,C 180,E1 -2121.299,E2 -2121.299} C_VEL
LIN {X 0,Y 573.242,Z 85.387,A -85,B 0,C 180,E1 -2124.015,E2 -2124.015} C_VEL
LIN {X 0,Y 573.273,Z 85.385,A -85,B 0,C 180,E1 -2126.518,E2 -2126.518} C_VEL
LIN {X 0,Y 573.232,Z 85.397,A -85,B 0,C 180,E1 -2129.118,E2 -2129.118} C_VEL
LIN {X 0,Y 573.24,Z 85.391,A -85,B 0,C 180,E1 -2131.436,E2 -2131.436} C_VEL
LIN {X 0,Y 573.263,Z 85.386,A -85,B 0,C 180,E1 -2133.81,E2 -2133.81} C_VEL
LIN {X 0,Y 573.24,Z 85.393,A -85,B 0,C 180,E1 -2136.381,E2 -2136.381} C_VEL
LIN {X 0,Y 574.586,Z 88.976,A -85,B 0,C 180,E1 -2136.493,E2 -2136.493} C_VEL
LIN {X 0,Y 576.172,Z 93.066,A -85,B 0,C 180,E1 -2136.619,E2 -2136.619} C_VEL
LIN {X 0,Y 575.501,Z 283.386,A -85,B 0,C 180,E1 -2139.118,E2 -2139.118} C_VEL
LIN {X 0,Y 575.383,Z 299.582,A -85,B 0,C 180,E1 -2139.441,E2 -2139.441} C_VEL
LIN {X 0,Y 575.2,Z 315.271,A -85,B 0,C 180,E1 -2139.901,E2 -2139.901} C_VEL
LIN {X 0,Y 574.998,Z 328.702,A -85,B 0,C 180,E1 -2140.404,E2 -2140.404} C_VEL
LIN {X 0,Y 574.758,Z 343.728,A -85,B 0,C 180,E1 -2141.093,E2 -2141.093} C_VEL
LIN {X 0,Y 574.436,Z 358.233,A -85,B 0,C 180,E1 -2141.913,E2 -2141.913} C_VEL
LIN {X 0,Y 574.192,Z 370.859,A -85,B 0,C 180,E1 -2142.76,E2 -2142.76} C_VEL
LIN {X 0,Y 573.948,Z 384.493,A -85,B 0,C 180,E1 -2143.825,E2 -2143.825} C_VEL
LIN {X 0,Y 573.716,Z 398.054,A -85,B 0,C 180,E1 -2145.093,E2 -2145.093} C_VEL
LIN {X 0,Y 573.505,Z 408.01,A -85,B 0,C 180,E1 -2146.175,E2 -2146.175} C_VEL
LIN {X 0,Y 573.358,Z 418.038,A -85,B 0,C 180,E1 -2147.433,E2 -2147.433} C_VEL
LIN {X 0,Y 573.256,Z 427.991,A -85,B 0,C 180,E1 -2148.898,E2 -2148.898} C_VEL
LIN {X 0,Y 573.113,Z 436.814,A -85,B 0,C 180,E1 -2150.471,E2 -2150.471} C_VEL
LIN {X 0,Y 573.057,Z 443.419,A -85,B 0,C 180,E1 -2151.892,E2 -2151.892} C_VEL
LIN {X 0,Y 573.031,Z 449.224,A -85,B 0,C 180,E1 -2153.433,E2 -2153.433} C_VEL
LIN {X 0,Y 572.946,Z 453.966,A -85,B 0,C 180,E1 -2155.074,E2 -2155.074} C_VEL
LIN {X 0,Y 573.006,Z 456.89,A -85,B 0,C 180,E1 -2156.484,E2 -2156.484} C_VEL
LIN {X 0,Y 572.927,Z 458.847,A -85,B 0,C 180,E1 -2157.891,E2 -2157.891} C_VEL
LIN {X 0,Y 572.939,Z 459.817,A -85,B 0,C 180,E1 -2159.297,E2 -2159.297} C_VEL
LIN {X 0,Y 572.94,Z 459.846,A -85,B 0,C 180,E1 -2160.703,E2 -2160.703} C_VEL
LIN {X 0,Y 572.927,Z 458.933,A -85,B 0,C 180,E1 -2162.109,E2 -2162.109} C_VEL
LIN {X 0,Y 573.005,Z 457.033,A -85,B 0,C 180,E1 -2163.516,E2 -2163.516} C_VEL
LIN {X 0,Y 572.944,Z 454.191,A -85,B 0,C 180,E1 -2164.926,E2 -2164.926} C_VEL
LIN {X 0,Y 573.032,Z 449.533,A -85,B 0,C 180,E1 -2166.568,E2 -2166.568} C_VEL
LIN {X 0,Y 573.057,Z 443.799,A -85,B 0,C 180,E1 -2168.108,E2 -2168.108} C_VEL
LIN {X 0,Y 573.107,Z 437.267,A -85,B 0,C 180,E1 -2169.529,E2 -2169.529} C_VEL
LIN {X 0,Y 573.202,Z 429.646,A -85,B 0,C 180,E1 -2170.919,E2 -2170.919} C_VEL
LIN {X 0,Y 573.334,Z 420.057,A -85,B 0,C 180,E1 -2172.387,E2 -2172.387} C_VEL
LIN {X 0,Y 573.498,Z 410.307,A -85,B 0,C 180,E1 -2173.645,E2 -2173.645} C_VEL
LIN {X 0,Y 573.636,Z 400.699,A -85,B 0,C 180,E1 -2174.724,E2 -2174.724} C_VEL
LIN {X 0,Y 573.82,Z 391.523,A -85,B 0,C 180,E1 -2175.631,E2 -2175.631} C_VEL
LIN {X 0,Y 574.056,Z 380.036,A -85,B 0,C 180,E1 -2176.629,E2 -2176.629} C_VEL
LIN {X 0,Y 574.295,Z 367.554,A -85,B 0,C 180,E1 -2177.565,E2 -2177.565} C_VEL
LIN {X 0,Y 574.572,Z 352.076,A -85,B 0,C 180,E1 -2178.543,E2 -2178.543} C_VEL
LIN {X 0,Y 574.816,Z 337.997,A -85,B 0,C 180,E1 -2179.276,E2 -2179.276} C_VEL
LIN {X 0,Y 575.104,Z 322.042,A -85,B 0,C 180,E1 -2179.954,E2 -2179.954} C_VEL
LIN {X 0,Y 575.332,Z 307.008,A -85,B 0,C 180,E1 -2180.444,E2 -2180.444} C_VEL
LIN {X 0,Y 575.427,Z 292.117,A -85,B 0,C 180,E1 -2180.814,E2 -2180.814} C_VEL
LIN {X 0,Y 575.593,Z 271.868,A -85,B 0,C 180,E1 -2181.135,E2 -2181.135} C_VEL
LIN {X 0,Y 576.108,Z 92.476,A -85,B 0,C 180,E1 -2183.481,E2 -2183.481} C_VEL
LIN {X 0,Y 573.372,Z 86.33,A -85,B 0,C 180,E1 -2183.687,E2 -2183.687} C_VEL
LIN {X 0,Y 573.205,Z 85.397,A -85,B 0,C 180,E1 -2183.721,E2 -2183.721} C_VEL
LIN {X 0,Y 573.199,Z 85.398,A -85,B 0,C 180,E1 -2186.484,E2 -2186.484} C_VEL
LIN {X 0,Y 573.227,Z 85.393,A -85,B 0,C 180,E1 -2189.368,E2 -2189.368} C_VEL
LIN {X 0,Y 573.24,Z 85.392,A -85,B 0,C 180,E1 -2192.226,E2 -2192.226} C_VEL
LIN {X 0,Y 573.233,Z 85.396,A -85,B 0,C 180,E1 -2194.77,E2 -2194.77} C_VEL
LIN {X 0,Y 573.229,Z 85.391,A -85,B 0,C 180,E1 -2197.808,E2 -2197.808} C_VEL
LIN {X 0,Y 573.247,Z 85.394,A -85,B 0,C 180,E1 -2200.525,E2 -2200.525} C_VEL
LIN {X 0,Y 573.232,Z 85.389,A -85,B 0,C 180,E1 -2203.359,E2 -2203.359} C_VEL
LIN {X 0,Y 573.249,Z 85.392,A -85,B 0,C 180,E1 -2206.33,E2 -2206.33} C_VEL
LIN {X 0,Y 573.232,Z 85.391,A -85,B 0,C 180,E1 -2208.543,E2 -2208.543} C_VEL
LIN {X 0,Y 573.243,Z 85.39,A -85,B 0,C 180,E1 -2211.298,E2 -2211.298} C_VEL
LIN {X 0,Y 573.214,Z 85.398,A -85,B 0,C 180,E1 -2214.018,E2 -2214.018} C_VEL
LIN {X 0,Y 573.287,Z 85.386,A -85,B 0,C 180,E1 -2216.519,E2 -2216.519} C_VEL
LIN {X 0,Y 573.229,Z 85.399,A -85,B 0,C 180,E1 -2219.117,E2 -2219.117} C_VEL
LIN {X 0,Y 573.265,Z 85.47,A -85,B 0,C 180,E1 -2220.577,E2 -2220.577} C_VEL
LIN {X 0,Y 575.738,Z 94.375,A -85,B 0,C 180,E1 -2221.392,E2 -2221.392} C_VEL
LIN {X 0,Y 575.442,Z 131.257,A -85,B 0,C 180,E1 -2224.237,E2 -2224.237} C_VEL
LIN {X 0,Y 575.198,Z 158.852,A -85,B 0,C 180,E1 -2226.341,E2 -2226.341} C_VEL
LIN {X 0,Y 576.203,Z 165.356,A -85,B 0,C 180,E1 -2226.471,E2 -2226.471} C_VEL
LIN {X 0,Y 575.496,Z 366.401,A -85,B 0,C 180,E1 -2229.118,E2 -2229.118} C_VEL
LIN {X 0,Y 575.366,Z 382.989,A -85,B 0,C 180,E1 -2229.487,E2 -2229.487} C_VEL
LIN {X 0,Y 575.136,Z 399.228,A -85,B 0,C 180,E1 -2229.992,E2 -2229.992} C_VEL
LIN {X 0,Y 574.884,Z 415.171,A -85,B 0,C 180,E1 -2230.637,E2 -2230.637} C_VEL
LIN {X 0,Y 574.662,Z 429.707,A -85,B 0,C 180,E1 -2231.367,E2 -2231.367} C_VEL
LIN {X 0,Y 574.363,Z 444.647,A -85,B 0,C 180,E1 -2232.277,E2 -2232.277} C_VEL
LIN {X 0,Y 574.054,Z 458.379,A -85,B 0,C 180,E1 -2233.279,E2 -2233.279} C_VEL
LIN {X 0,Y 573.831,Z 471.064,A -85,B 0,C 180,E1 -2234.368,E2 -2234.368} C_VEL
LIN {X 0,Y 573.605,Z 483.276,A -85,B 0,C 180,E1 -2235.595,E2 -2235.595} C_VEL
LIN {X 0,Y 573.419,Z 494.333,A -85,B 0,C 180,E1 -2236.894,E2 -2236.894} C_VEL
LIN {X 0,Y 573.283,Z 504.669,A -85,B 0,C 180,E1 -2238.329,E2 -2238.329} C_VEL
LIN {X 0,Y 573.169,Z 513.282,A -85,B 0,C 180,E1 -2239.758,E2 -2239.758} C_VEL
LIN {X 0,Y 573.077,Z 520.487,A -85,B 0,C 180,E1 -2241.182,E2 -2241.182} C_VEL
LIN {X 0,Y 573.039,Z 526.465,A -85,B 0,C 180,E1 -2242.601,E2 -2242.601} C_VEL
LIN {X 0,Y 573.017,Z 531.185,A -85,B 0,C 180,E1 -2244.015,E2 -2244.015} C_VEL
LIN {X 0,Y 573.005,Z 535.636,A -85,B 0,C 180,E1 -2245.779,E2 -2245.779} C_VEL
LIN {X 0,Y 572.949,Z 538.088,A -85,B 0,C 180,E1 -2247.187,E2 -2247.187} C_VEL
LIN {X 0,Y 572.943,Z 539.479,A -85,B 0,C 180,E1 -2248.594,E2 -2248.594} C_VEL
LIN {X 0,Y 572.933,Z 540,A -85,B 0,C 180,E1 -2250,E2 -2250} C_VEL
LIN {X 0,Y 572.943,Z 539.48,A -85,B 0,C 180,E1 -2251.405,E2 -2251.405} C_VEL
LIN {X 0,Y 572.948,Z 538.089,A -85,B 0,C 180,E1 -2252.812,E2 -2252.812} C_VEL
LIN {X 0,Y 573.005,Z 535.637,A -85,B 0,C 180,E1 -2254.22,E2 -2254.22} C_VEL
LIN {X 0,Y 573.015,Z 531.189,A -85,B 0,C 180,E1 -2255.984,E2 -2255.984} C_VEL
LIN {X 0,Y 573.041,Z 526.47,A -85,B 0,C 180,E1 -2257.398,E2 -2257.398} C_VEL
LIN {X 0,Y 573.093,Z 518.859,A -85,B 0,C 180,E1 -2259.173,E2 -2259.173} C_VEL
LIN {X 0,Y 573.151,Z 511.267,A -85,B 0,C 180,E1 -2260.598,E2 -2260.598} C_VEL
LIN {X 0,Y 573.303,Z 502.216,A -85,B 0,C 180,E1 -2262.028,E2 -2262.028} C_VEL
LIN {X 0,Y 573.442,Z 491.427,A -85,B 0,C 180,E1 -2263.465,E2 -2263.465} C_VEL
LIN {X 0,Y 573.656,Z 480.304,A -85,B 0,C 180,E1 -2264.725,E2 -2264.725} C_VEL
LIN {X 0,Y 573.901,Z 468.147,A -85,B 0,C 180,E1 -2265.902,E2 -2265.902} C_VEL
LIN {X 0,Y 574.131,Z 454.879,A -85,B 0,C 180,E1 -2266.993,E2 -2266.993} C_VEL
LIN {X 0,Y 574.431,Z 441.859,A -85,B 0,C 180,E1 -2267.902,E2 -2267.902} C_VEL
LIN {X 0,Y 574.665,Z 428.036,A -85,B 0,C 180,E1 -2268.725,E2 -2268.725} C_VEL
